(* Logix 5000 project; controller VET 1756-L62 rev 19.52; software revision 19.01; part 5 of 27 *)

        [443].S.BITS1.10   // 110-ENF-001/2 LH
        [444].S.BITS1.0   // 110-ENF-001/2-1 Enable
        [444].S.BITS1.1   // 110-ENF-001/2-1 Falla Resumen
        [444].S.BITS1.2   // 110-ENF-001/2-1 Conf. Marcha
        [444].S.BITS1.4   // 110-ENF-001/2-1 Cmd. Automatico
        [444].S.BITS1.26   // 110-ENF-001/2-1 FLL
        [444].S.BITS1.28   // 110-ENF-001/2-1 FATO
        [444].S.BITS1.30   // 110-ENF-001/2-1 Falla Partida
        [444].S.BITS2.27   // 110-ENF-001/2-1 Cmd. Marcha
        [444].S.BITS2.20   // 110-ENF-001/2-1 Reset Falla
        [444].S.BITS2.23   // 110-ENF-001/2-1 Test
        [444].S.BITS2.30   // 110-ENF-001/2-1 OUT MARCHA
        [447].S.BITS1.27   // 110-ESC-003/2 FV0
        [446].S.BITS1.8   // 9-BIN-708 LL
        [446].S.BITS1.9   // 9-BIN-708 LM
        [446].S.BITS1.10   // 9-BIN-708 LH
        [447].S.BITS1.0   // 9-CON-709 Enable
        [447].S.BITS1.1   // 9-CON-709 Falla Resumen
        [447].S.BITS1.26   // 110-ESC-003/2 FLL
        [447].S.BITS1.28   // 110-ESC-003/2 FATO
        [447].S.BITS2.20   // 9-CON-709 Reset Falla
        [447].S.BITS2.23   // 9-CON-709 Test
        [447].S.BITS2.30   // 9-CON-709 OUT CLOSE
        [449].S.BITS1.0   // 9-CON-711 Enable
        [449].S.BITS1.1   // 9-CON-711 Falla Resumen
        [449].S.BITS1.4   // 9-CON-711 Conf Pos Cerrar
        [449].S.BITS1.26   // 110-VAL-001/2-1 FLL
        [449].S.BITS1.27   // 110-VAL-001/2-1 FV0
        [449].S.BITS1.28   // 110-VAL-001/2-1 FATO
        [449].S.BITS2.20   // 9-CON-711 Reset Falla
        [449].S.BITS2.23   // 9-CON-711 Test
        [449].S.BITS2.30   // 9-CON-711 OUT CLOSE
        [450].S.BITS1.0   // 110-VEN-001/2 Enable
        [450].S.BITS1.1   // 110-VEN-001/2 Falla Resumen
        [450].S.BITS1.2   // 110-VEN-001/2 Conf. Marcha
        [450].S.BITS1.4   // 110-VEN-001/2 Cmd. Automatico
        [450].S.BITS1.26   // 110-VEN-001/2 FLL
        [450].S.BITS1.27   // 110-VEN-001/2 FV0
        [450].S.BITS1.28   // 110-VEN-001/2 FATO
        [450].S.BITS1.30   // 110-VEN-001/2 Falla Partida
        [450].S.BITS2.27   // 110-VEN-001/2 Cmd. Marcha
        [450].S.BITS2.20   // 110-VEN-001/2 Reset Falla
        [450].S.BITS2.23   // 110-VEN-001/2 Test
        [450].S.BITS2.30   // 110-VEN-001/2 OUT MARCHA
        [451].S.BITS1.0   // 9-CON-713 Enable
        [451].S.BITS1.1   // 9-CON-713 Falla Resumen
        [451].S.BITS1.2   // 9-CON-713 Conf Pos Abrir
        [451].S.BITS1.4   // 9-CON-713 Conf Pos Cerrar
        [451].S.BITS1.26   // 110-ENF-001/2-5 FLL
        [451].S.BITS1.27   // 110-ENF-001/2-5 FV0
        [451].S.BITS1.28   // 110-ENF-001/2-5 FATO
        [451].S.BITS1.30   // 9-CON-713 Falla Cerrar
        [451].S.BITS2.27   // 9-CON-713 Cmd. Open
        [451].S.BITS2.20   // 9-CON-713 Reset Falla
        [451].S.BITS2.23   // 9-CON-713 Test
        [451].S.BITS2.30   // 9-CON-713 OUT CLOSE
        [461].S.BITS1.0   // 9-CON-723 Enable
        [461].S.BITS1.1   // 9-CON-723 Falla Resumen
        [461].S.BITS1.2   // 9-CON-723 Conf Pos Abrir
        [461].S.BITS1.4   // 9-CON-723 Conf Pos Cerrar
        [461].S.BITS1.26   // 110-ESC-002/2 FLL
        [461].S.BITS1.27   // 110-ESC-002/2 FV0
        [461].S.BITS1.28   // 110-ESC-002/2 FATO
        [461].S.BITS1.30   // 9-CON-723 Falla Cerrar
        [461].S.BITS2.27   // 9-CON-723 Cmd. Open
        [461].S.BITS2.20   // 9-CON-723 Reset Falla
        [461].S.BITS2.23   // 9-CON-723 Test
        [461].S.BITS2.30   // 9-CON-723 OUT CLOSE
        [462].S.BITS1.0   // 110-ENF-002/2-4 Enable
        [462].S.BITS1.1   // 110-ENF-002/2-4 Falla Resumen
        [462].S.BITS1.2   // 110-ENF-002/2-4 Conf. Marcha
        [462].S.BITS1.4   // 110-ENF-002/2-4 Cmd. Automatico
        [462].S.BITS1.26   // 110-ENF-002/2-4 FLL
        [462].S.BITS1.27   // 110-ENF-002/2-4 FV0
        [462].S.BITS1.28   // 110-ENF-002/2-4 FATO
        [462].S.BITS1.30   // 110-ENF-002/2-4 Falla Partida
        [462].S.BITS2.27   // 110-ENF-002/2-4 Cmd. Marcha
        [462].S.BITS2.20   // 110-ENF-002/2-4 Reset Falla
        [462].S.BITS2.23   // 110-ENF-002/2-4 Test
        [462].S.BITS2.30   // 110-ENF-002/2-4 OUT MARCHA
        [464].S.BITS1.27   // 110-ENF-002/2-1 FV0
        [463].S.BITS1.8   // 110-ENF-002/2 LL
        [463].S.BITS1.9   // 110-ENF-002/2 LM
        [463].S.BITS1.10   // 110-ENF-002/2 LH
        [464].S.BITS1.0   // 110-ENF-002/2-1 Enable
        [464].S.BITS1.1   // 110-ENF-002/2-1 Falla Resumen
        [464].S.BITS1.2   // 110-ENF-002/2-1 Conf. Marcha
        [464].S.BITS1.4   // 110-ENF-002/2-1 Cmd. Automatico
        [464].S.BITS1.26   // 110-ENF-002/2-1 FLL
        [464].S.BITS1.28   // 110-ENF-002/2-1 FATO
        [464].S.BITS1.30   // 110-ENF-002/2-1 Falla Partida
        [464].S.BITS2.27   // 110-ENF-002/2-1 Cmd. Marcha
        [464].S.BITS2.20   // 110-ENF-002/2-1 Reset Falla
        [464].S.BITS2.23   // 110-ENF-002/2-1 Test
        [464].S.BITS2.30   // 110-ENF-002/2-1 OUT MARCHA
        [467].S.BITS1.27   // 110-ESC-004/2 FV0
        [466].S.BITS1.8   // 9-BIN-728 LL
        [466].S.BITS1.9   // 9-BIN-728 LM
        [466].S.BITS1.10   // 9-BIN-728 LH
        [467].S.BITS1.0   // 9-CON-729 Enable
        [467].S.BITS1.1   // 9-CON-729 Falla Resumen
        [467].S.BITS1.2   // 9-CON-729 Conf Pos Abrir
        [467].S.BITS1.4   // 9-CON-729 Conf Pos Cerrar
        [467].S.BITS1.26   // 110-ESC-004/2 FLL
        [467].S.BITS1.28   // 110-ESC-004/2 FATO
        [467].S.BITS1.30   // 9-CON-729 Falla Cerrar
        [467].S.BITS2.27   // 9-CON-729 Cmd. Open
        [467].S.BITS2.20   // 9-CON-729 Reset Falla
        [467].S.BITS2.23   // 9-CON-729 Test
        [467].S.BITS2.30   // 9-CON-729 OUT CLOSE
        [469].S.BITS1.0   // 9-CON-731 Enable
        [469].S.BITS1.1   // 9-CON-731 Falla Resumen
        [469].S.BITS1.2   // 9-CON-731 Conf Pos Abrir
        [469].S.BITS1.4   // 9-CON-731 Conf Pos Cerrar
        [469].S.BITS1.26   // 110-VAL-002/2-1 FLL
        [469].S.BITS1.27   // 110-VAL-002/2-1 FV0
        [469].S.BITS1.28   // 110-VAL-002/2-1 FATO
        [469].S.BITS1.30   // 9-CON-731 Falla Cerrar
        [469].S.BITS2.27   // 9-CON-731 Cmd. Open
        [469].S.BITS2.20   // 9-CON-731 Reset Falla
        [469].S.BITS2.23   // 9-CON-731 Test
        [469].S.BITS2.30   // 9-CON-731 OUT CLOSE
        [470].S.BITS1.0   // 110-VEN-002/2 Enable
        [470].S.BITS1.1   // 110-VEN-002/2 Falla Resumen
        [470].S.BITS1.2   // 110-VEN-002/2 Conf. Marcha
        [470].S.BITS1.4   // 110-VEN-002/2 Cmd. Automatico
        [470].S.BITS1.26   // 110-VEN-002/2 FLL
        [470].S.BITS1.27   // 110-VEN-002/2 FV0
        [470].S.BITS1.28   // 110-VEN-002/2 FATO
        [470].S.BITS1.30   // 110-VEN-002/2 Falla Partida
        [470].S.BITS2.27   // 110-VEN-002/2 Cmd. Marcha
        [470].S.BITS2.20   // 110-VEN-002/2 Reset Falla
        [470].S.BITS2.23   // 110-VEN-002/2 Test
        [470].S.BITS2.30   // 110-VEN-002/2 OUT MARCHA
        [471].S.BITS1.0   // 110-ENF-002/2-5 Enable
        [471].S.BITS1.1   // 110-ENF-002/2-5 Falla Resumen
        [471].S.BITS1.2   // 110-ENF-002/2-5 Conf. Marcha
        [471].S.BITS1.4   // 110-ENF-002/2-5 Cmd. Automatico
        [471].S.BITS1.26   // 110-ENF-002/2-5 FLL
        [471].S.BITS1.27   // 110-ENF-002/2-5 FV0
        [471].S.BITS1.28   // 110-ENF-002/2-5 FATO
        [471].S.BITS1.30   // 110-ENF-002/2-5 Falla Partida
        [471].S.BITS2.27   // 110-ENF-002/2-5 Cmd. Marcha
        [471].S.BITS2.20   // 110-ENF-002/2-5 Reset Falla
        [471].S.BITS2.23   // 110-ENF-002/2-5 Test
        [471].S.BITS2.30   // 110-ENF-002/2-5 OUT MARCHA
        [474].S.BITS1.0   // 110-TOR-002/2 Enable
        [474].S.BITS1.1   // 110-TOR-002/2 Falla Resumen
        [474].S.BITS1.26   // 110-TOR-002/2 FLL
        [474].S.BITS1.27   // 110-TOR-002/2 FV0
        [474].S.BITS1.28   // 110-TOR-002/2 FATO
        [474].S.BITS2.20   // 110-TOR-002/2 Reset Falla
        [474].S.BITS2.23   // 110-TOR-002/2 Test
        [474].S.BITS2.30   // 110-TOR-002/2 OUT MARCHA
        [475].S.BITS1.0   // 110-TOR-003/2 Enable
        [475].S.BITS1.1   // 110-TOR-003/2 Falla Resumen
        [475].S.BITS1.26   // 110-TOR-003/2 FLL
        [475].S.BITS1.27   // 110-TOR-003/2 FV0
        [475].S.BITS1.28   // 110-TOR-003/2 FATO
        [475].S.BITS2.20   // 110-TOR-003/2 Reset Falla
        [475].S.BITS2.23   // 110-TOR-003/2 Test
        [475].S.BITS2.30   // 110-TOR-003/2 OUT MARCHA
        [476].S.BITS1.0   // 110-ELV-002/2 Enable
        [476].S.BITS1.1   // 110-ELV-002/2 Falla Resumen
        [476].S.BITS1.26   // 110-ELV-002/2 FLL
        [476].S.BITS1.27   // 110-ELV-002/2 FV0
        [476].S.BITS1.28   // 110-ELV-002/2 FATO
        [476].S.BITS2.20   // 110-ELV-002/2 Reset Falla
        [476].S.BITS2.23   // 110-ELV-002/2 Test
        [478].S.BITS1.27   // 110-TOR-004/2 FV0
        [477].S.BITS1.8   // 110-TOL-006/2 LL
        [477].S.BITS1.9   // 110-TOL-006/2 LM
        [477].S.BITS1.10   // 110-TOL-006/2 LH
        [478].S.BITS1.0   // 110-TOR-004/2 Enable
        [478].S.BITS1.1   // 110-TOR-004/2 Falla Resumen
        [478].S.BITS1.2   // 110-TOR-004/2 Conf. Marcha
        [478].S.BITS1.4   // 110-TOR-004/2 Cmd. Automatico
        [478].S.BITS1.26   // 110-TOR-004/2 FLL
        [478].S.BITS1.28   // 110-TOR-004/2 FATO
        [478].S.BITS1.30   // 110-TOR-004/2 Falla Partida
        [478].S.BITS2.27   // 110-TOR-004/2 Cmd. Marcha
        [478].S.BITS2.20   // 110-TOR-004/2 Reset Falla
        [478].S.BITS2.23   // 110-TOR-004/2 Test
        [478].S.BITS2.30   // 110-TOR-004/2 OUT MARCHA
        [493].S.BITS1.1   // 110-CAN-008/3 Falla Resumen
        [491].S.BITS1.8   // 110-TOL-005/3 LL
        [491].S.BITS1.9   // 110-TOL-005/3 LM
        [491].S.BITS1.10   // 110-TOL-005/3 LH
        [493].S.BITS1.30   // 110-CAN-008/3 Falla Cerrar
        [492].S.BITS1.8   // 110-TOL-004/3 LL
        [492].S.BITS1.9   // 110-TOL-004/3 LM
        [492].S.BITS1.10   // 110-TOL-004/3 LH
        [493].S.BITS1.0   // 110-CAN-008/3 Enable
        [493].S.BITS1.2   // 110-CAN-008/3 Conf Pos Abrir
        [493].S.BITS1.4   // 110-CAN-008/3 Conf Pos Cerrar
        [493].S.BITS1.29   // 110-CAN-008/3 Falla Abrir
        [493].S.BITS2.20   // 110-CAN-008/3 Reset Falla
        [493].S.BITS2.23   // 110-CAN-008/3 Test
        [493].S.BITS2.27   // 110-CAN-008/3 Cmd. Open
        [493].S.BITS2.30   // 110-CAN-008/3 OUT CLOSE
        [493].S.BITS2.31   // 110-CAN-008/3 OUT OPEN
        [494].S.BITS1.0   // 110-CAN-009/3 Enable
        [494].S.BITS1.1   // 110-CAN-009/3 Falla Resumen
        [494].S.BITS1.2   // 110-CAN-009/3 Conf Pos Abrir
        [494].S.BITS1.4   // 110-CAN-009/3 Conf Pos Cerrar
        [494].S.BITS1.29   // 110-CAN-009/3 Falla Abrir
        [494].S.BITS1.30   // 110-CAN-009/3 Falla Cerrar
        [494].S.BITS2.20   // 110-CAN-009/3 Reset Falla
        [494].S.BITS2.23   // 110-CAN-009/3 Test
        [494].S.BITS2.27   // 110-CAN-009/3 Cmd. Open
        [494].S.BITS2.30   // 110-CAN-009/3 OUT CLOSE
        [494].S.BITS2.31   // 110-CAN-009/3 OUT OPEN
        [495].S.BITS1.0   // 110-CAN-010/3 Enable
        [495].S.BITS1.1   // 110-CAN-010/3 Falla Resumen
        [495].S.BITS1.2   // 110-CAN-010/3 Conf. Marcha
        [495].S.BITS1.4   // 110-CAN-010/3 Cmd. Automatico
        [495].S.BITS1.26   // 110-CAN-010/3 FLL
        [495].S.BITS1.27   // 110-CAN-010/3 FV0
        [495].S.BITS1.28   // 110-CAN-010/3 FATO
        [495].S.BITS1.30   // 110-CAN-010/3 Falla Partida
        [495].S.BITS2.27   // 110-CAN-010/3 Cmd. Marcha
        [495].S.BITS2.20   // 110-CAN-010/3 Reset Falla
        [495].S.BITS2.23   // 110-CAN-010/3 Test
        [495].S.BITS2.30   // 110-CAN-010/3 OUT MARCHA
        [497].S.BITS1.30   // 110-CAN-011/3 Falla Cerrar
        [496].S.BITS1.8   // 110-TOL-006/3 LL
        [496].S.BITS1.9   // 110-TOL-006/3 LM
        [496].S.BITS1.10   // 110-TOL-006/3 LH
        [497].S.BITS1.0   // 110-CAN-011/3 Enable
        [497].S.BITS1.1   // 110-CAN-011/3 Falla Resumen
        [497].S.BITS1.2   // 110-CAN-011/3 Conf Pos Abrir
        [497].S.BITS1.4   // 110-CAN-011/3 Conf Pos Cerrar
        [497].S.BITS1.29   // 110-CAN-011/3 Falla Abrir
        [497].S.BITS2.20   // 110-CAN-011/3 Reset Falla
        [497].S.BITS2.23   // 110-CAN-011/3 Test
        [497].S.BITS2.27   // 110-CAN-011/3 Cmd. Open
        [497].S.BITS2.30   // 110-CAN-011/3 OUT CLOSE
        [497].S.BITS2.31   // 110-CAN-011/3 OUT OPEN
        [500].S.BITS1.27   // 110-TOR-001/3 FV0
        [499].S.BITS1.8   // 110-TOL-007/3 LL
        [499].S.BITS1.9   // 110-TOL-007/3 LM
        [499].S.BITS1.10   // 110-TOL-007/3 LH
        [500].S.BITS1.0   // 110-TOR-001/3 Enable
        [500].S.BITS1.1   // 110-TOR-001/3 Falla Resumen
        [500].S.BITS1.2   // 110-TOR-001/3 Conf. Marcha
        [500].S.BITS1.4   // 110-TOR-001/3 Cmd. Automatico
        [500].S.BITS1.26   // 110-TOR-001/3 FLL
        [500].S.BITS1.28   // 110-TOR-001/3 FATO
        [500].S.BITS1.30   // 110-TOR-001/3 Falla Partida
        [500].S.BITS2.27   // 110-TOR-001/3 Cmd. Marcha
        [500].S.BITS2.20   // 110-TOR-001/3 Reset Falla
        [500].S.BITS2.23   // 110-TOR-001/3 Test
        [500].S.BITS2.30   // 110-TOR-001/3 OUT MARCHA
        [502].S.BITS1.0   // 110-ACD-001/3 Enable
        [502].S.BITS1.1   // 110-ACD-001/3 Falla Resumen
        [502].S.BITS1.2   // 110-ACD-001/3 Conf. Marcha
        [502].S.BITS1.4   // 110-ACD-001/3 Cmd. Automatico
        [502].S.BITS1.26   // 110-ACD-001/3 FLL
        [502].S.BITS1.27   // 110-ACD-001/3 FV0
        [502].S.BITS1.28   // 110-ACD-001/3 FATO
        [502].S.BITS1.30   // 110-ACD-001/3 Falla Partida
        [502].S.BITS2.27   // 110-ACD-001/3 Cmd. Marcha
        [502].S.BITS2.20   // 110-ACD-001/3 Reset Falla
        [502].S.BITS2.23   // 110-ACD-001/3 Test
        [502].S.BITS2.30   // 110-ACD-001/3 OUT MARCHA
        [503].S.BITS1.0   // 110-EXP-001/3 Enable
        [503].S.BITS1.1   // 110-EXP-001/3 Falla Resumen
        [503].S.BITS1.4   // 110-EXP-001/3 Cmd. Automatico
        [503].S.BITS1.26   // 110-EXP-001/3 FLL
        [503].S.BITS1.27   // 110-EXP-001/3 FV0
        [503].S.BITS1.28   // 110-EXP-001/3 FATO
        [503].S.BITS1.30   // 110-EXP-001/3 Falla Partida
        [503].S.BITS2.27   // 110-EXP-001/3 Cmd. Marcha
        [503].S.BITS2.20   // 110-EXP-001/3 Reset Falla
        [503].S.BITS2.23   // 110-EXP-001/3 Test
        [503].S.BITS2.30   // 110-EXP-001/3 OUT MARCHA
        [504].S.BITS1.0   // 110-DES-001/3 Enable
        [504].S.BITS1.1   // 110-DES-001/3 Falla Resumen
        [504].S.BITS1.2   // 110-DES-001/3 Conf. Marcha
        [504].S.BITS1.4   // 110-DES-001/3 Cmd. Automatico
        [504].S.BITS1.26   // 110-DES-001/3 FLL
        [504].S.BITS1.27   // 110-DES-001/3 FV0
        [504].S.BITS1.28   // 110-DES-001/3 FATO
        [504].S.BITS1.30   // 110-DES-001/3 Falla Partida
        [504].S.BITS2.27   // 110-DES-001/3 Cmd. Marcha
        [504].S.BITS2.20   // 110-DES-001/3 Reset Falla
        [504].S.BITS2.23   // 110-DES-001/3 Test
        [504].S.BITS2.30   // 110-DES-001/3 OUT MARCHA
        [505].S.BITS1.0   // 110-CAE-001/3 Enable
        [505].S.BITS1.1   // 110-CAE-001/3 Falla Resumen
        [505].S.BITS1.2   // 110-CAE-001/3 Conf. Marcha
        [505].S.BITS1.4   // 110-CAE-001/3 Cmd. Automatico
        [505].S.BITS1.26   // 110-CAE-001/3 FLL
        [505].S.BITS1.27   // 110-CAE-001/3 FV0
        [505].S.BITS1.28   // 110-CAE-001/3 FATO
        [505].S.BITS1.30   // 110-CAE-001/3 Falla Partida
        [505].S.BITS2.27   // 110-CAE-001/3 Cmd. Marcha
        [505].S.BITS2.20   // 110-CAE-001/3 Reset Falla
        [505].S.BITS2.23   // 110-CAE-001/3 Test
        [505].S.BITS2.30   // 110-CAE-001/3 OUT MARCHA
        [506].S.BITS1.0   // 110-PLT-001/3 Enable
        [506].S.BITS1.1   // 110-PLT-001/3 Falla Resumen
        [506].S.BITS1.2   // 110-PLT-001/3 Conf. Marcha
        [506].S.BITS1.4   // 110-PLT-001/3 Cmd. Automatico
        [506].S.BITS1.26   // 110-PLT-001/3 FLL
        [506].S.BITS1.27   // 110-PLT-001/3 FV0
        [506].S.BITS1.28   // 110-PLT-001/3 FATO
        [506].S.BITS1.30   // 110-PLT-001/3 Falla Partida
        [506].S.BITS2.27   // 110-PLT-001/3 Cmd. Marcha
        [506].S.BITS2.20   // 110-PLT-001/3 Reset Falla
        [506].S.BITS2.23   // 110-PLT-001/3 Test
        [506].S.BITS2.30   // 110-PLT-001/3 OUT MARCHA
        [507].S.BITS1.0   // 110-BIF-001/3 Enable
        [507].S.BITS1.1   // 110-BIF-001/3 Falla Resumen
        [507].S.BITS1.2   // 110-BIF-001/3 Conf. Pos. Izquierda
        [507].S.BITS1.4   // 110-BIF-001/3 Conf. Pos. Derecha
        [507].S.BITS1.29   // 110-BIF-001/3 Falla Pos. Izquierda
        [507].S.BITS1.30   // 110-BIF-001/3 Falla Pos. Derecha
        [507].S.BITS2.20   // 110-BIF-001/3 Reset Falla
        [507].S.BITS2.23   // 110-BIF-001/3 Test
        [507].S.BITS2.26   // 110-BIF-001/3 Cmd. Pos . Izquierda
        [507].S.BITS2.27   // 110-BIF-001/3 Cmd. Pos. Derecha
        [507].S.BITS2.30   // 110-BIF-001/3 Out Izquierda
        [507].S.BITS2.31   // 110-BIF-001/3 Out Derecha
        [511].S.BITS1.0   // 110-ESC-001/3 Enable
        [511].S.BITS1.1   // 110-ESC-001/3 Falla Resumen
        [511].S.BITS1.2   // 110-ESC-001/3 Conf. Marcha
        [511].S.BITS1.4   // 110-ESC-001/3 Cmd. Automatico
        [511].S.BITS1.26   // 110-ESC-001/3 FLL
        [511].S.BITS1.27   // 110-ESC-001/3 FV0
        [511].S.BITS1.28   // 110-ESC-001/3 FATO
        [511].S.BITS1.30   // 110-ESC-001/3 Falla Partida
        [511].S.BITS2.27   // 110-ESC-001/3 Cmd. Marcha
        [511].S.BITS2.20   // 110-ESC-001/3 Reset Falla
        [511].S.BITS2.23   // 110-ESC-001/3 Test
        [511].S.BITS2.30   // 110-ESC-001/3 OUT MARCHA
        [512].S.BITS1.0   // 110-ENF-001/3-4 Enable
        [512].S.BITS1.1   // 110-ENF-001/3-4 Falla Resumen
        [512].S.BITS1.2   // 110-ENF-001/3-4 Conf. Marcha
        [512].S.BITS1.4   // 110-ENF-001/3-4 Cmd. Automatico
        [512].S.BITS1.26   // 110-ENF-001/3-4 FLL
        [512].S.BITS1.27   // 110-ENF-001/3-4 FV0
        [512].S.BITS1.28   // 110-ENF-001/3-4 FATO
        [512].S.BITS1.30   // 110-ENF-001/3-4 Falla Partida
        [512].S.BITS2.27   // 110-ENF-001/3-4 Cmd. Marcha
        [512].S.BITS2.20   // 110-ENF-001/3-4 Reset Falla
        [512].S.BITS2.23   // 110-ENF-001/3-4 Test
        [512].S.BITS2.30   // 110-ENF-001/3-4 OUT MARCHA
        [514].S.BITS1.27   // 110-ENF-001/3-1 FV0
        [513].S.BITS1.8   // 110-ENF-001/3 LL
        [513].S.BITS1.9   // 110-ENF-001/3 LM
        [513].S.BITS1.10   // 110-ENF-001/3 LH
        [514].S.BITS1.0   // 110-ENF-001/3-1 Enable
        [514].S.BITS1.1   // 110-ENF-001/3-1 Falla Resumen
        [514].S.BITS1.2   // 110-ENF-001/3-1 Conf. Marcha
        [514].S.BITS1.4   // 110-ENF-001/3-1 Cmd. Automatico
        [514].S.BITS1.26   // 110-ENF-001/3-1 FLL
        [514].S.BITS1.28   // 110-ENF-001/3-1 FATO
        [514].S.BITS1.30   // 110-ENF-001/3-1 Falla Partida
        [514].S.BITS2.27   // 110-ENF-001/3-1 Cmd. Marcha
        [514].S.BITS2.20   // 110-ENF-001/3-1 Reset Falla
        [514].S.BITS2.23   // 110-ENF-001/3-1 Test
        [514].S.BITS2.30   // 110-ENF-001/3-1 OUT MARCHA
        [517].S.BITS1.27   // 110-ESC-003/3 FV0
        [516].S.BITS1.8   // 110-CIC-001/3 LL
        [516].S.BITS1.9   // 110-CIC-001/3 LM
        [516].S.BITS1.10   // 110-CIC-001/3 LH
        [517].S.BITS1.0   // 110-ESC-003/3 Enable
        [517].S.BITS1.1   // 110-ESC-003/3 Falla Resumen
        [517].S.BITS1.2   // 110-ESC-003/3 Conf. Marcha
        [517].S.BITS1.4   // 110-ESC-003/3 Cmd. Automatico
        [517].S.BITS1.26   // 110-ESC-003/3 FLL
        [517].S.BITS1.28   // 110-ESC-003/3 FATO
        [517].S.BITS1.30   // 110-ESC-003/3 Falla Partida
        [517].S.BITS2.27   // 110-ESC-003/3 Cmd. Marcha
        [517].S.BITS2.20   // 110-ESC-003/3 Reset Falla
        [517].S.BITS2.23   // 110-ESC-003/3 Test
        [517].S.BITS2.30   // 110-ESC-003/3 OUT MARCHA
        [519].S.BITS1.0   // 110-VAL-001/3-1 Enable
        [519].S.BITS1.1   // 110-VAL-001/3-1 Falla Resumen
        [519].S.BITS1.2   // 110-VAL-001/3-1 Conf. Marcha
        [519].S.BITS1.4   // 110-VAL-001/3-1 Cmd. Automatico
        [519].S.BITS1.26   // 110-VAL-001/3-1 FLL
        [519].S.BITS1.27   // 110-VAL-001/3-1 FV0
        [519].S.BITS1.28   // 110-VAL-001/3-1 FATO
        [519].S.BITS1.30   // 110-VAL-001/3-1 Falla Partida
        [519].S.BITS2.27   // 110-VAL-001/3-1 Cmd. Marcha
        [519].S.BITS2.20   // 110-VAL-001/3-1 Reset Falla
        [519].S.BITS2.23   // 110-VAL-001/3-1 Test
        [519].S.BITS2.30   // 110-VAL-001/3-1 OUT MARCHA
        [520].S.BITS1.0   // 110-VEN-001/3 Enable
        [520].S.BITS1.1   // 110-VEN-001/3 Falla Resumen
        [520].S.BITS1.2   // 110-VEN-001/3 Conf. Marcha
        [520].S.BITS1.4   // 110-VEN-001/3 Cmd. Automatico
        [520].S.BITS1.26   // 110-VEN-001/3 FLL
        [520].S.BITS1.27   // 110-VEN-001/3 FV0
        [520].S.BITS1.28   // 110-VEN-001/3 FATO
        [520].S.BITS1.30   // 110-VEN-001/3 Falla Partida
        [520].S.BITS2.27   // 110-VEN-001/3 Cmd. Marcha
        [520].S.BITS2.20   // 110-VEN-001/3 Reset Falla
        [520].S.BITS2.23   // 110-VEN-001/3 Test
        [520].S.BITS2.30   // 110-VEN-001/3 OUT MARCHA
        [521].S.BITS1.0   // 110-ENF-001/3-5 Enable
        [521].S.BITS1.1   // 110-ENF-001/3-5 Falla Resumen
        [521].S.BITS1.2   // 110-ENF-001/3-5 Conf. Marcha
        [521].S.BITS1.4   // 110-ENF-001/3-5 Cmd. Automatico
        [521].S.BITS1.26   // 110-ENF-001/3-5 FLL
        [521].S.BITS1.27   // 110-ENF-001/3-5 FV0
        [521].S.BITS1.28   // 110-ENF-001/3-5 FATO
        [521].S.BITS1.30   // 110-ENF-001/3-5 Falla Partida
        [521].S.BITS2.27   // 110-ENF-001/3-5 Cmd. Marcha
        [521].S.BITS2.20   // 110-ENF-001/3-5 Reset Falla
        [521].S.BITS2.23   // 110-ENF-001/3-5 Test
        [521].S.BITS2.30   // 110-ENF-001/3-5 OUT MARCHA
        [523].S.BITS1.0   // 110-QUE-001-1 Enable
        [523].S.BITS1.1   // 110-QUE-001-1 Falla Resumen
        [523].S.BITS1.2   // 110-QUE-001-1 Conf. Marcha
        [523].S.BITS1.4   // 110-QUE-001-1 Cmd. Automatico
        [523].S.BITS1.26   // 110-QUE-001-1 FLL
        [523].S.BITS1.27   // 110-QUE-001-1 FV0
        [523].S.BITS1.28   // 110-QUE-001-1 FATO
        [523].S.BITS1.30   // 110-QUE-001-1 Falla Partida
        [523].S.BITS2.27   // 110-QUE-001-1 Cmd. Marcha
        [523].S.BITS2.20   // 110-QUE-001-1 Reset Falla
        [523].S.BITS2.23   // 110-QUE-001-1 Test
        [523].S.BITS2.30   // 110-QUE-001-1 OUT MARCHA
        [524].S.BITS1.0   // 110-QUE-001-2 Enable
        [524].S.BITS1.1   // 110-QUE-001-2 Falla Resumen
        [524].S.BITS1.2   // 110-QUE-001-2 Conf. Marcha
        [524].S.BITS1.4   // 110-QUE-001-2 Cmd. Automatico
        [524].S.BITS1.26   // 110-QUE-001-2 FLL
        [524].S.BITS1.27   // 110-QUE-001-2 FV0
        [524].S.BITS1.28   // 110-QUE-001-2 FATO
        [524].S.BITS1.30   // 110-QUE-001-2 Falla Partida
        [524].S.BITS2.27   // 110-QUE-001-2 Cmd. Marcha
        [524].S.BITS2.20   // 110-QUE-001-2 Reset Falla
        [524].S.BITS2.23   // 110-QUE-001-2 Test
        [524].S.BITS2.30   // 110-QUE-001-2 OUT MARCHA
        [531].S.BITS1.0   // 110-ESC-002/3 Enable
        [531].S.BITS1.1   // 110-ESC-002/3 Falla Resumen
        [531].S.BITS1.2   // 110-ESC-002/3 Conf. Marcha
        [531].S.BITS1.4   // 110-ESC-002/3 Cmd. Automatico
        [531].S.BITS1.26   // 110-ESC-002/3 FLL
        [531].S.BITS1.27   // 110-ESC-002/3 FV0
        [531].S.BITS1.28   // 110-ESC-002/3 FATO
        [531].S.BITS1.30   // 110-ESC-002/3 Falla Partida
        [531].S.BITS2.27   // 110-ESC-002/3 Cmd. Marcha
        [531].S.BITS2.20   // 110-ESC-002/3 Reset Falla
        [531].S.BITS2.23   // 110-ESC-002/3 Test
        [531].S.BITS2.30   // 110-ESC-002/3 OUT MARCHA
        [532].S.BITS1.0   // 110-ENF-002/3-4 Enable
        [532].S.BITS1.1   // 110-ENF-002/3-4 Falla Resumen
        [532].S.BITS1.2   // 110-ENF-002/3-4 Conf. Marcha
        [532].S.BITS1.4   // 110-ENF-002/3-4 Cmd. Automatico
        [532].S.BITS1.26   // 110-ENF-002/3-4 FLL
        [532].S.BITS1.27   // 110-ENF-002/3-4 FV0
        [532].S.BITS1.28   // 110-ENF-002/3-4 FATO
        [532].S.BITS1.30   // 110-ENF-002/3-4 Falla Partida
        [532].S.BITS2.27   // 110-ENF-002/3-4 Cmd. Marcha
        [532].S.BITS2.20   // 110-ENF-002/3-4 Reset Falla
        [532].S.BITS2.23   // 110-ENF-002/3-4 Test
        [532].S.BITS2.30   // 110-ENF-002/3-4 OUT MARCHA
        [534].S.BITS1.27   // 110-ENF-002/3-1 FV0
        [533].S.BITS1.8   // 110-ENF-002/3 LL
        [533].S.BITS1.9   // 110-ENF-002/3 LM
        [533].S.BITS1.10   // 110-ENF-002/3 LH
        [534].S.BITS1.0   // 110-ENF-002/3-1 Enable
        [534].S.BITS1.1   // 110-ENF-002/3-1 Falla Resumen
        [534].S.BITS1.2   // 110-ENF-002/3-1 Conf. Marcha
        [534].S.BITS1.4   // 110-ENF-002/3-1 Cmd. Automatico
        [534].S.BITS1.26   // 110-ENF-002/3-1 FLL
        [534].S.BITS1.28   // 110-ENF-002/3-1 FATO
        [534].S.BITS1.30   // 110-ENF-002/3-1 Falla Partida
        [534].S.BITS2.27   // 110-ENF-002/3-1 Cmd. Marcha
        [534].S.BITS2.20   // 110-ENF-002/3-1 Reset Falla
        [534].S.BITS2.23   // 110-ENF-002/3-1 Test
        [534].S.BITS2.30   // 110-ENF-002/3-1 OUT MARCHA
        [537].S.BITS1.27   // 110-ESC-004/3 FV0
        [536].S.BITS1.8   // 110-CIC-002/3 LL
        [536].S.BITS1.9   // 110-CIC-002/3 LM
        [536].S.BITS1.10   // 110-CIC-002/3 LH
        [537].S.BITS1.0   // 110-ESC-004/3 Enable
        [537].S.BITS1.1   // 110-ESC-004/3 Falla Resumen
        [537].S.BITS1.2   // 110-ESC-004/3 Conf. Marcha
        [537].S.BITS1.4   // 110-ESC-004/3 Cmd. Automatico
        [537].S.BITS1.26   // 110-ESC-004/3 FLL
        [537].S.BITS1.28   // 110-ESC-004/3 FATO
        [537].S.BITS1.30   // 110-ESC-004/3 Falla Partida
        [537].S.BITS2.27   // 110-ESC-004/3 Cmd. Marcha
        [537].S.BITS2.20   // 110-ESC-004/3 Reset Falla
        [537].S.BITS2.23   // 110-ESC-004/3 Test
        [537].S.BITS2.30   // 110-ESC-004/3 OUT MARCHA
        [539].S.BITS1.0   // 110-VEN-002/3-1 Enable
        [539].S.BITS1.1   // 110-VEN-002/3-1 Falla Resumen
        [539].S.BITS1.2   // 110-VEN-002/3-1 Conf. Marcha
        [539].S.BITS1.4   // 110-VEN-002/3-1 Cmd. Automatico
        [539].S.BITS1.26   // 110-VEN-002/3-1 FLL
        [539].S.BITS1.27   // 110-VEN-002/3-1 FV0
        [539].S.BITS1.28   // 110-VEN-002/3-1 FATO
        [539].S.BITS1.30   // 110-VEN-002/3-1 Falla Partida
        [539].S.BITS2.27   // 110-VEN-002/3-1 Cmd. Marcha
        [539].S.BITS2.20   // 110-VEN-002/3-1 Reset Falla
        [539].S.BITS2.23   // 110-VEN-002/3-1 Test
        [539].S.BITS2.30   // 110-VEN-002/3-1 OUT MARCHA
        [540].S.BITS1.0   // 110-VEN-002/3 Enable
        [540].S.BITS1.1   // 110-VEN-002/3 Falla Resumen
        [540].S.BITS1.2   // 110-VEN-002/3 Conf. Marcha
        [540].S.BITS1.4   // 110-VEN-002/3 Cmd. Automatico
        [540].S.BITS1.26   // 110-VEN-002/3 FLL
        [540].S.BITS1.27   // 110-VEN-002/3 FV0
        [540].S.BITS1.28   // 110-VEN-002/3 FATO
        [540].S.BITS1.30   // 110-VEN-002/3 Falla Partida
        [540].S.BITS2.27   // 110-VEN-002/3 Cmd. Marcha
        [540].S.BITS2.20   // 110-VEN-002/3 Reset Falla
        [540].S.BITS2.23   // 110-VEN-002/3 Test
        [540].S.BITS2.30   // 110-VEN-002/3 OUT MARCHA
        [541].S.BITS1.0   // 110-ENF-002/3-5 Enable
        [541].S.BITS1.1   // 110-ENF-002/3-5 Falla Resumen
        [541].S.BITS1.2   // 110-ENF-002/3-5 Conf. Marcha
        [541].S.BITS1.4   // 110-ENF-002/3-5 Cmd. Automatico
        [541].S.BITS1.26   // 110-ENF-002/3-5 FLL
        [541].S.BITS1.27   // 110-ENF-002/3-5 FV0
        [541].S.BITS1.28   // 110-ENF-002/3-5 FATO
        [541].S.BITS1.30   // 110-ENF-002/3-5 Falla Partida
        [541].S.BITS2.27   // 110-ENF-002/3-5 Cmd. Marcha
        [541].S.BITS2.20   // 110-ENF-002/3-5 Reset Falla
        [541].S.BITS2.23   // 110-ENF-002/3-5 Test
        [541].S.BITS2.30   // 110-ENF-002/3-5 OUT MARCHA
        [544].S.BITS1.0   // 110-TOR-002/3 Enable
        [544].S.BITS1.1   // 110-TOR-002/3 Falla Resumen
        [544].S.BITS1.2   // 110-TOR-002/3 Conf. Marcha
        [544].S.BITS1.4   // 110-TOR-002/3 Cmd. Automatico
        [544].S.BITS1.26   // 110-TOR-002/3 FLL
        [544].S.BITS1.27   // 110-TOR-002/3 FV0
        [544].S.BITS1.28   // 110-TOR-002/3 FATO
        [544].S.BITS1.30   // 110-TOR-002/3 Falla Partida
        [544].S.BITS2.27   // 110-TOR-002/3 Cmd. Marcha
        [544].S.BITS2.20   // 110-TOR-002/3 Reset Falla
        [544].S.BITS2.23   // 110-TOR-002/3 Test
        [544].S.BITS2.30   // 110-TOR-002/3 OUT MARCHA
        [545].S.BITS1.0   // 110-TOR-003/3 Enable
        [545].S.BITS1.1   // 110-TOR-003/3 Falla Resumen
        [545].S.BITS1.2   // 110-TOR-003/3 Conf. Marcha
        [545].S.BITS1.4   // 110-TOR-003/3 Cmd. Automatico
        [545].S.BITS1.26   // 110-TOR-003/3 FLL
        [545].S.BITS1.27   // 110-TOR-003/3 FV0
        [545].S.BITS1.28   // 110-TOR-003/3 FATO
        [545].S.BITS1.30   // 110-TOR-003/3 Falla Partida
        [545].S.BITS2.27   // 110-TOR-003/3 Cmd. Marcha
        [545].S.BITS2.20   // 110-TOR-003/3 Reset Falla
        [545].S.BITS2.23   // 110-TOR-003/3 Test
        [545].S.BITS2.30   // 110-TOR-003/3 OUT MARCHA
        [546].S.BITS1.0   // 110-ELV-002/3 Enable
        [546].S.BITS1.1   // 110-ELV-002/3 Falla Resumen
        [546].S.BITS1.2   // 110-ELV-002/3 Conf. Marcha
        [546].S.BITS1.4   // 110-ELV-002/3 Cmd. Automatico
        [546].S.BITS1.26   // 110-ELV-002/3 FLL
        [546].S.BITS1.27   // 110-ELV-002/3 FV0
        [546].S.BITS1.28   // 110-ELV-002/3 FATO
        [546].S.BITS1.30   // 110-ELV-002/3 Falla Partida
        [546].S.BITS2.27   // 110-ELV-002/3 Cmd. Marcha
        [546].S.BITS2.20   // 110-ELV-002/3 Reset Falla
        [546].S.BITS2.23   // 110-ELV-002/3 Test
        [546].S.BITS2.30   // 110-ELV-002/3 OUT MARCHA
        [548].S.BITS1.27   // 110-TOR-004/3 FV0
        [547].S.BITS1.8   // 110-TOL-008/3 LL
        [547].S.BITS1.9   // 110-TOL-008/3 LM
        [547].S.BITS1.10   // 110-TOL-008/3 LH
        [548].S.BITS1.0   // 110-TOR-004/3 Enable
        [548].S.BITS1.1   // 110-TOR-004/3 Falla Resumen
        [548].S.BITS1.2   // 110-TOR-004/3 Conf. Marcha
        [548].S.BITS1.4   // 110-TOR-004/3 Cmd. Automatico
        [548].S.BITS1.26   // 110-TOR-004/3 FLL
        [548].S.BITS1.28   // 110-TOR-004/3 FATO
        [548].S.BITS1.30   // 110-TOR-004/3 Falla Partida
        [548].S.BITS2.27   // 110-TOR-004/3 Cmd. Marcha
        [548].S.BITS2.20   // 110-TOR-004/3 Reset Falla
        [548].S.BITS2.23   // 110-TOR-004/3 Test
        [548].S.BITS2.30   // 110-TOR-004/3 OUT MARCHA
        [551].S.BITS1.0   // 110-TDC-003/1 Enable
        [551].S.BITS1.1   // 110-TDC-003/1 Falla Resumen
        [551].S.BITS1.2   // 110-TDC-003/1 Conf. Marcha
        [551].S.BITS1.4   // 110-TDC-003/1 Cmd. Automatico
        [551].S.BITS1.26   // 110-TDC-003/1 FLL
        [551].S.BITS1.27   // 110-TDC-003/1 FV0
        [551].S.BITS1.28   // 110-TDC-003/1 FATO
        [551].S.BITS1.30   // 110-TDC-003/1 Falla Partida
        [551].S.BITS2.27   // 110-TDC-003/1 Cmd. Marcha
        [551].S.BITS2.20   // 110-TDC-003/1 Reset Falla
        [551].S.BITS2.23   // 110-TDC-003/1 Test
        [551].S.BITS2.30   // 110-TDC-003/1 OUT MARCHA
        [552].S.BITS1.26   // 110-TDC-004/1 FLL
        [552].S.BITS1.27   // 110-TDC-004/1 FV0
        [552].S.BITS1.28   // 110-TDC-004/1 FATO
        [554].S.BITS1.26   // 110-ELV-001/1 FLL
        [554].S.BITS1.27   // 110-ELV-001/1 FV0
        [554].S.BITS1.28   // 110-ELV-001/1 FATO
        [555].S.BITS1.0   // 120-TDC-001/1 Enable
        [555].S.BITS1.1   // 120-TDC-001/1 Falla Resumen
        [555].S.BITS1.2   // 120-TDC-001/1 Conf. Marcha
        [555].S.BITS1.4   // 120-TDC-001/1 Cmd. Automatico
        [555].S.BITS1.26   // 120-TDC-001/1 FLL
        [555].S.BITS1.27   // 120-TDC-001/1 FV0
        [555].S.BITS1.28   // 120-TDC-001/1 FATO
        [555].S.BITS1.30   // 120-TDC-001/1 Falla Partida
        [555].S.BITS2.27   // 120-TDC-001/1 Cmd. Marcha
        [555].S.BITS2.20   // 120-TDC-001/1 Reset Falla
        [555].S.BITS2.23   // 120-TDC-001/1 Test
        [555].S.BITS2.30   // 120-TDC-001/1 OUT MARCHA
        [556].S.BITS1.26   // 120-HAR-001 FLL
        [556].S.BITS1.27   // 120-HAR-001 FV0
        [556].S.BITS1.28   // 120-HAR-001 FATO
        [557].S.BITS1.0   // 120-XY-8127 Enable
        [557].S.BITS1.1   // 120-XY-8127 Falla Resumen
        [557].S.BITS1.2   // 120-XY-8127 Conf Pos Abrir
        [557].S.BITS1.4   // 120-XY-8127 Conf Pos Cerrar
        [557].S.BITS1.29   // 120-XY-8127 Falla Abrir
        [557].S.BITS1.30   // 120-XY-8127 Falla Cerrar
        [557].S.BITS2.20   // 120-XY-8127 Reset Falla
        [557].S.BITS2.23   // 120-XY-8127 Test
        [557].S.BITS2.27   // 120-XY-8127 Cmd. Open
        [557].S.BITS2.30   // 120-XY-8127 OUT CLOSE
        [557].S.BITS2.31   // 120-XY-8127 OUT OPEN
        [558].S.BITS1.0   // 120-TDC-002 Enable
        [558].S.BITS1.1   // 120-TDC-002 Falla Resumen
        [558].S.BITS1.2   // 120-TDC-002 Conf. Marcha
        [558].S.BITS1.4   // 120-TDC-002 Cmd. Automatico
        [558].S.BITS1.26   // 120-TDC-002 FLL
        [558].S.BITS1.27   // 120-TDC-002 FV0
        [558].S.BITS1.28   // 120-TDC-002 FATO
        [558].S.BITS1.30   // 120-TDC-002 Falla Partida
        [558].S.BITS2.27   // 120-TDC-002 Cmd. Marcha
        [558].S.BITS2.20   // 120-TDC-002 Reset Falla
        [558].S.BITS2.23   // 120-TDC-002 Test
        [558].S.BITS2.30   // 120-TDC-002 OUT MARCHA
        [559].S.BITS1.0   // 120-CAN-001 Enable
        [559].S.BITS1.1   // 120-CAN-001 Falla Resumen
        [559].S.BITS1.2   // 120-CAN-001 Conf Pos Abrir
        [559].S.BITS1.4   // 120-CAN-001 Conf Pos Cerrar
        [559].S.BITS1.29   // 120-CAN-001 Falla Abrir
        [559].S.BITS1.30   // 120-CAN-001 Falla Cerrar
        [559].S.BITS2.20   // 120-CAN-001 Reset Falla
        [559].S.BITS2.23   // 120-CAN-001 Test
        [559].S.BITS2.27   // 120-CAN-001 Cmd. Open
        [559].S.BITS2.30   // 120-CAN-001 OUT CLOSE
        [559].S.BITS2.31   // 120-CAN-001 OUT OPEN
        [561].S.BITS1.0   // 110-TDC-003/2 Enable
        [561].S.BITS1.1   // 110-TDC-003/2 Falla Resumen
        [561].S.BITS1.2   // 110-TDC-003/2 Conf. Marcha
        [561].S.BITS1.4   // 110-TDC-003/2 Cmd. Automatico
        [561].S.BITS1.26   // 110-TDC-003/2 FLL
        [561].S.BITS1.27   // 110-TDC-003/2 FV0
        [561].S.BITS1.28   // 110-TDC-003/2 FATO
        [561].S.BITS1.30   // 110-TDC-003/2 Falla Partida
        [561].S.BITS2.27   // 110-TDC-003/2 Cmd. Marcha
        [561].S.BITS2.20   // 110-TDC-003/2 Reset Falla
        [561].S.BITS2.23   // 110-TDC-003/2 Test
        [561].S.BITS2.30   // 110-TDC-003/2 OUT MARCHA
        [562].S.BITS1.0   // 110-TDC-004/2 Enable
        [562].S.BITS1.1   // 110-TDC-004/2 Falla Resumen
        [562].S.BITS1.2   // 110-TDC-004/2 Conf. Marcha
        [562].S.BITS1.4   // 110-TDC-004/2 Cmd. Automatico
        [562].S.BITS1.26   // 110-TDC-004/2 FLL
        [562].S.BITS1.27   // 110-TDC-004/2 FV0
        [562].S.BITS1.28   // 110-TDC-004/2 FATO
        [562].S.BITS1.30   // 110-TDC-004/2 Falla Partida
        [562].S.BITS2.27   // 110-TDC-004/2 Cmd. Marcha
        [562].S.BITS2.20   // 110-TDC-004/2 Reset Falla
        [562].S.BITS2.23   // 110-TDC-004/2 Test
        [562].S.BITS2.30   // 110-TDC-004/2 OUT MARCHA
        [564].S.BITS1.0   // 110-ELV-001/2 Enable
        [564].S.BITS1.1   // 110-ELV-001/2 Falla Resumen
        [564].S.BITS1.2   // 110-ELV-001/2 Conf. Marcha
        [564].S.BITS1.4   // 110-ELV-001/2 Cmd. Automatico
        [564].S.BITS1.26   // 110-ELV-001/2 FLL
        [564].S.BITS1.27   // 110-ELV-001/2 FV0
        [564].S.BITS1.28   // 110-ELV-001/2 FATO
        [564].S.BITS1.30   // 110-ELV-001/2 Falla Partida
        [564].S.BITS2.27   // 110-ELV-001/2 Cmd. Marcha
        [564].S.BITS2.20   // 110-ELV-001/2 Reset Falla
        [564].S.BITS2.23   // 110-ELV-001/2 Test
        [564].S.BITS2.30   // 110-ELV-001/2 OUT MARCHA
        [565].S.BITS1.0   // 120-TDC-001/2 Enable
        [565].S.BITS1.1   // 120-TDC-001/2 Falla Resumen
        [565].S.BITS1.2   // 120-TDC-001/2 Conf. Marcha
        [565].S.BITS1.4   // 120-TDC-001/2 Cmd. Automatico
        [565].S.BITS1.26   // 120-TDC-001/2 FLL
        [565].S.BITS1.27   // 120-TDC-001/2 FV0
        [565].S.BITS1.28   // 120-TDC-001/2 FATO
        [565].S.BITS1.30   // 120-TDC-001/2 Falla Partida
        [565].S.BITS2.27   // 120-TDC-001/2 Cmd. Marcha
        [565].S.BITS2.20   // 120-TDC-001/2 Reset Falla
        [565].S.BITS2.23   // 120-TDC-001/2 Test
        [565].S.BITS2.30   // 120-TDC-001/2 OUT MARCHA
        [566].S.BITS1.0   // 120-HAR-002 Enable
        [566].S.BITS1.1   // 120-HAR-002 Falla Resumen
        [566].S.BITS1.2   // 120-HAR-002 Conf. Marcha
        [566].S.BITS1.4   // 120-HAR-002 Cmd. Automatico
        [566].S.BITS1.26   // 120-HAR-002 FLL
        [566].S.BITS1.27   // 120-HAR-002 FV0
        [566].S.BITS1.28   // 120-HAR-002 FATO
        [566].S.BITS1.30   // 120-HAR-002 Falla Partida
        [566].S.BITS2.27   // 120-HAR-002 Cmd. Marcha
        [566].S.BITS2.20   // 120-HAR-002 Reset Falla
        [566].S.BITS2.23   // 120-HAR-002 Test
        [566].S.BITS2.30   // 120-HAR-002 OUT MARCHA
        [567].S.BITS1.0   // 120-XY-8128 Enable
        [567].S.BITS1.1   // 120-XY-8128 Falla Resumen
        [567].S.BITS1.2   // 120-XY-8128 Conf Pos Abrir
        [567].S.BITS1.4   // 120-XY-8128 Conf Pos Cerrar
        [567].S.BITS1.29   // 120-XY-8128 Falla Abrir
        [567].S.BITS1.30   // 120-XY-8128 Falla Cerrar
        [567].S.BITS2.20   // 120-XY-8128 Reset Falla
        [567].S.BITS2.23   // 120-XY-8128 Test
        [567].S.BITS2.27   // 120-XY-8128 Cmd. Open
        [567].S.BITS2.30   // 120-XY-8128 OUT CLOSE
        [567].S.BITS2.31   // 120-XY-8128 OUT OPEN
        [568].S.BITS1.0   // 120-TDC-003 Enable
        [568].S.BITS1.1   // 120-TDC-003 Falla Resumen
        [568].S.BITS1.2   // 120-TDC-003 Conf. Marcha
        [568].S.BITS1.4   // 120-TDC-003 Cmd. Automatico
        [568].S.BITS1.26   // 120-TDC-003 FLL
        [568].S.BITS1.27   // 120-TDC-003 FV0
        [568].S.BITS1.28   // 120-TDC-003 FATO
        [568].S.BITS1.30   // 120-TDC-003 Falla Partida
        [568].S.BITS2.27   // 120-TDC-003 Cmd. Marcha
        [568].S.BITS2.20   // 120-TDC-003 Reset Falla
        [568].S.BITS2.23   // 120-TDC-003 Test
        [568].S.BITS2.30   // 120-TDC-003 OUT MARCHA
        [569].S.BITS1.0   // 120-CAN-003 Enable
        [569].S.BITS1.1   // 120-CAN-003 Falla Resumen
        [569].S.BITS1.2   // 120-CAN-003 Conf Pos Abrir
        [569].S.BITS1.4   // 120-CAN-003 Conf Pos Cerrar
        [569].S.BITS1.29   // 120-CAN-003 Falla Abrir
        [569].S.BITS1.30   // 120-CAN-003 Falla Cerrar
        [569].S.BITS2.20   // 120-CAN-003 Reset Falla
        [569].S.BITS2.23   // 120-CAN-003 Test
        [569].S.BITS2.27   // 120-CAN-003 Cmd. Open
        [569].S.BITS2.30   // 120-CAN-003 OUT CLOSE
        [569].S.BITS2.31   // 120-CAN-003 OUT OPEN
        [571].S.BITS1.0   // 110-TDC-003/3 Enable
        [571].S.BITS1.1   // 110-TDC-003/3 Falla Resumen
        [571].S.BITS1.2   // 110-TDC-003/3 Conf. Marcha
        [571].S.BITS1.4   // 110-TDC-003/3 Cmd. Automatico
        [571].S.BITS1.26   // 110-TDC-003/3 FLL
        [571].S.BITS1.27   // 110-TDC-003/3 FV0
        [571].S.BITS1.28   // 110-TDC-003/3 FATO
        [571].S.BITS1.30   // 110-TDC-003/3 Falla Partida
        [571].S.BITS2.27   // 110-TDC-003/3 Cmd. Marcha
        [571].S.BITS2.20   // 110-TDC-003/3 Reset Falla
        [571].S.BITS2.23   // 110-TDC-003/3 Test
        [571].S.BITS2.30   // 110-TDC-003/3 OUT MARCHA
        [572].S.BITS1.0   // 110-TDC-004/3 Enable
        [572].S.BITS1.1   // 110-TDC-004/3 Falla Resumen
        [572].S.BITS1.2   // 110-TDC-004/3 Conf. Marcha
        [572].S.BITS1.4   // 110-TDC-004/3 Cmd. Automatico
        [572].S.BITS1.26   // 110-TDC-004/3 FLL
        [572].S.BITS1.27   // 110-TDC-004/3 FV0
        [572].S.BITS1.28   // 110-TDC-004/3 FATO
        [572].S.BITS1.30   // 110-TDC-004/3 Falla Partida
        [572].S.BITS2.27   // 110-TDC-004/3 Cmd. Marcha
        [572].S.BITS2.20   // 110-TDC-004/3 Reset Falla
        [572].S.BITS2.23   // 110-TDC-004/3 Test
        [572].S.BITS2.30   // 110-TDC-004/3 OUT MARCHA
        [573].S.BITS1.0   // 110-TDC-005/3 Enable
        [573].S.BITS1.1   // 110-TDC-005/3 Falla Resumen
        [573].S.BITS1.2   // 110-TDC-005/3 Conf. Marcha
        [573].S.BITS1.4   // 110-TDC-005/3 Cmd. Automatico
        [573].S.BITS1.26   // 110-TDC-005/3 FLL
        [573].S.BITS1.27   // 110-TDC-005/3 FV0
        [573].S.BITS1.28   // 110-TDC-005/3 FATO
        [573].S.BITS1.30   // 110-TDC-005/3 Falla Partida
        [573].S.BITS2.27   // 110-TDC-005/3 Cmd. Marcha
        [573].S.BITS2.20   // 110-TDC-005/3 Reset Falla
        [573].S.BITS2.23   // 110-TDC-005/3 Test
        [573].S.BITS2.30   // 110-TDC-005/3 OUT MARCHA
        [574].S.BITS1.0   // 110-ELV-001/3 Enable
        [574].S.BITS1.1   // 110-ELV-001/3 Falla Resumen
        [574].S.BITS1.2   // 110-ELV-001/3 Conf. Marcha
        [574].S.BITS1.4   // 110-ELV-001/3 Cmd. Automatico
        [574].S.BITS1.26   // 110-ELV-001/3 FLL
        [574].S.BITS1.27   // 110-ELV-001/3 FV0
        [574].S.BITS1.28   // 110-ELV-001/3 FATO
        [574].S.BITS1.30   // 110-ELV-001/3 Falla Partida
        [574].S.BITS2.27   // 110-ELV-001/3 Cmd. Marcha
        [574].S.BITS2.20   // 110-ELV-001/3 Reset Falla
        [574].S.BITS2.23   // 110-ELV-001/3 Test
        [574].S.BITS2.30   // 110-ELV-001/3 OUT MARCHA
        [575].S.BITS1.0   // 120-TDC-001/3 Enable
        [575].S.BITS1.1   // 120-TDC-001/3 Falla Resumen
        [575].S.BITS1.2   // 120-TDC-001/3 Conf. Marcha
        [575].S.BITS1.4   // 120-TDC-001/3 Cmd. Automatico
        [575].S.BITS1.26   // 120-TDC-001/3 FLL
        [575].S.BITS1.27   // 120-TDC-001/3 FV0
        [575].S.BITS1.28   // 120-TDC-001/3 FATO
        [575].S.BITS1.30   // 120-TDC-001/3 Falla Partida
        [575].S.BITS2.27   // 120-TDC-001/3 Cmd. Marcha
        [575].S.BITS2.20   // 120-TDC-001/3 Reset Falla
        [575].S.BITS2.23   // 120-TDC-001/3 Test
        [575].S.BITS2.30   // 120-TDC-001/3 OUT MARCHA
        [576].S.BITS1.0   // 120-HAR-003 Enable
        [576].S.BITS1.1   // 120-HAR-003 Falla Resumen
        [576].S.BITS1.2   // 120-HAR-003 Conf. Marcha
        [576].S.BITS1.4   // 120-HAR-003 Cmd. Automatico
        [576].S.BITS1.26   // 120-HAR-003 FLL
        [576].S.BITS1.27   // 120-HAR-003 FV0
        [576].S.BITS1.28   // 120-HAR-003 FATO
        [576].S.BITS1.30   // 120-HAR-003 Falla Partida
        [576].S.BITS2.27   // 120-HAR-003 Cmd. Marcha
        [576].S.BITS2.20   // 120-HAR-003 Reset Falla
        [576].S.BITS2.23   // 120-HAR-003 Test
        [576].S.BITS2.30   // 120-HAR-003 OUT MARCHA
        [577].S.BITS1.0   // 120-XY-8129 Enable
        [577].S.BITS1.1   // 120-XY-8129 Falla Resumen
        [577].S.BITS1.2   // 120-XY-8129 Conf Pos Abrir
        [577].S.BITS1.4   // 120-XY-8129 Conf Pos Cerrar
        [577].S.BITS1.29   // 120-XY-8129 Falla Abrir
        [577].S.BITS1.30   // 120-XY-8129 Falla Cerrar
        [577].S.BITS2.20   // 120-XY-8129 Reset Falla
        [577].S.BITS2.23   // 120-XY-8129 Test
        [577].S.BITS2.27   // 120-XY-8129 Cmd. Open
        [577].S.BITS2.30   // 120-XY-8129 OUT CLOSE
        [577].S.BITS2.31   // 120-XY-8129 OUT OPEN
        [578].S.BITS1.0   // 120-BIF-001 Enable
        [578].S.BITS1.1   // 120-BIF-001 Falla Resumen
        [578].S.BITS1.2   // 120-BIF-001 Conf. Pos. Izquierda
        [578].S.BITS1.4   // 120-BIF-001 Conf. Pos. Derecha
        [578].S.BITS1.29   // 120-BIF-001 Falla Pos. Izquierda
        [578].S.BITS1.30   // 120-BIF-001 Falla Pos. Derecha
        [578].S.BITS2.20   // 120-BIF-001 Reset Falla
        [578].S.BITS2.23   // 120-BIF-001 Test
        [578].S.BITS2.26   // 120-BIF-001 Cmd. Pos . Izquierda
        [578].S.BITS2.27   // 120-BIF-001 Cmd. Pos. Derecha
        [578].S.BITS2.30   // 120-BIF-001 Out Izquierda
        [578].S.BITS2.31   // 120-BIF-001 Out Derecha
        [581].S.BITS1.0   // 120-TDC-005 Enable
        [581].S.BITS1.1   // 120-TDC-005 Falla Resumen
        [581].S.BITS1.2   // 120-TDC-005 Conf. Marcha
        [581].S.BITS1.4   // 120-TDC-005 Cmd. Automatico
        [581].S.BITS1.26   // 120-TDC-005 FLL
        [581].S.BITS1.27   // 120-TDC-005 FV0
        [581].S.BITS1.28   // 120-TDC-005 FATO
        [581].S.BITS1.30   // 120-TDC-005 Falla Partida
        [581].S.BITS2.27   // 120-TDC-005 Cmd. Marcha
        [581].S.BITS2.20   // 120-TDC-005 Reset Falla
        [581].S.BITS2.23   // 120-TDC-005 Test
        [581].S.BITS2.30   // 120-TDC-005 OUT MARCHA
        [582].S.BITS1.0   // 120-CAN-007 Enable
        [582].S.BITS1.1   // 120-CAN-007 Falla Resumen
        [582].S.BITS1.2   // 120-CAN-007 Conf Pos Abrir
        [582].S.BITS1.4   // 120-CAN-007 Conf Pos Cerrar
        [582].S.BITS1.29   // 120-CAN-007 Falla Abrir
        [582].S.BITS1.30   // 120-CAN-007 Falla Cerrar
        [582].S.BITS2.20   // 120-CAN-007 Reset Falla
        [582].S.BITS2.23   // 120-CAN-007 Test
        [582].S.BITS2.27   // 120-CAN-007 Cmd. Open
        [582].S.BITS2.30   // 120-CAN-007 OUT CLOSE
        [582].S.BITS2.31   // 120-CAN-007 OUT OPEN
        [583].S.BITS1.0   // 120-CAN-008 Enable
        [583].S.BITS1.1   // 120-CAN-008 Falla Resumen
        [583].S.BITS1.2   // 120-CAN-008 Conf Pos Abrir
        [583].S.BITS1.4   // 120-CAN-008 Conf Pos Cerrar
        [583].S.BITS1.29   // 120-CAN-008 Falla Abrir
        [583].S.BITS1.30   // 120-CAN-008 Falla Cerrar
        [583].S.BITS2.20   // 120-CAN-008 Reset Falla
        [583].S.BITS2.23   // 120-CAN-008 Test
        [583].S.BITS2.27   // 120-CAN-008 Cmd. Open
        [583].S.BITS2.30   // 120-CAN-008 OUT CLOSE
        [583].S.BITS2.31   // 120-CAN-008 OUT OPEN
        [584].S.BITS1.0   // 120-CAN-009 Enable
        [584].S.BITS1.1   // 120-CAN-009 Falla Resumen
        [584].S.BITS1.2   // 120-CAN-009 Conf Pos Abrir
        [584].S.BITS1.4   // 120-CAN-009 Conf Pos Cerrar
        [584].S.BITS1.29   // 120-CAN-009 Falla Abrir
        [584].S.BITS1.30   // 120-CAN-009 Falla Cerrar
        [584].S.BITS2.20   // 120-CAN-009 Reset Falla
        [584].S.BITS2.23   // 120-CAN-009 Test
        [584].S.BITS2.27   // 120-CAN-009 Cmd. Open
        [584].S.BITS2.30   // 120-CAN-009 OUT CLOSE
        [584].S.BITS2.31   // 120-CAN-009 OUT OPEN
        [585].S.BITS1.0   // 120-CAN-010 Enable
        [585].S.BITS1.1   // 120-CAN-010 Falla Resumen
        [585].S.BITS1.2   // 120-CAN-010 Conf Pos Abrir
        [585].S.BITS1.4   // 120-CAN-010 Conf Pos Cerrar
        [585].S.BITS1.29   // 120-CAN-010 Falla Abrir
        [585].S.BITS1.30   // 120-CAN-010 Falla Cerrar
        [585].S.BITS2.20   // 120-CAN-010 Reset Falla
        [585].S.BITS2.23   // 120-CAN-010 Test
        [585].S.BITS2.27   // 120-CAN-010 Cmd. Open
        [585].S.BITS2.30   // 120-CAN-010 OUT CLOSE
        [585].S.BITS2.31   // 120-CAN-010 OUT OPEN
        [586].S.BITS1.0   // 120-CAN-011 Enable
        [586].S.BITS1.1   // 120-CAN-011 Falla Resumen
        [586].S.BITS1.2   // 120-CAN-011 Conf Pos Abrir
        [586].S.BITS1.4   // 120-CAN-011 Conf Pos Cerrar
        [586].S.BITS1.29   // 120-CAN-011 Falla Abrir
        [586].S.BITS1.30   // 120-CAN-011 Falla Cerrar
        [586].S.BITS2.20   // 120-CAN-011 Reset Falla
        [586].S.BITS2.23   // 120-CAN-011 Test
        [586].S.BITS2.27   // 120-CAN-011 Cmd. Open
        [586].S.BITS2.30   // 120-CAN-011 OUT CLOSE
        [586].S.BITS2.31   // 120-CAN-011 OUT OPEN
        [587].S.BITS1.0   // 120-CAN-012 Enable
        [587].S.BITS1.1   // 120-CAN-012 Falla Resumen
        [587].S.BITS1.2   // 120-CAN-012 Conf Pos Abrir
        [587].S.BITS1.4   // 120-CAN-012 Conf Pos Cerrar
        [587].S.BITS1.29   // 120-CAN-012 Falla Abrir
        [587].S.BITS1.30   // 120-CAN-012 Falla Cerrar
        [587].S.BITS2.20   // 120-CAN-012 Reset Falla
        [587].S.BITS2.23   // 120-CAN-012 Test
        [587].S.BITS2.27   // 120-CAN-012 Cmd. Open
        [587].S.BITS2.30   // 120-CAN-012 OUT CLOSE
        [587].S.BITS2.31   // 120-CAN-012 OUT OPEN
        [588].S.BITS1.0   // 120-CAN-013 Enable
        [588].S.BITS1.1   // 120-CAN-013 Falla Resumen
        [588].S.BITS1.2   // 120-CAN-013 Conf Pos Abrir
        [588].S.BITS1.4   // 120-CAN-013 Conf Pos Cerrar
        [588].S.BITS1.29   // 120-CAN-013 Falla Abrir
        [588].S.BITS1.30   // 120-CAN-013 Falla Cerrar
        [588].S.BITS2.20   // 120-CAN-013 Reset Falla
        [588].S.BITS2.23   // 120-CAN-013 Test
        [588].S.BITS2.27   // 120-CAN-013 Cmd. Open
        [588].S.BITS2.30   // 120-CAN-013 OUT CLOSE
        [588].S.BITS2.31   // 120-CAN-013 OUT OPEN
        [589].S.BITS1.0   // 120-CAN-014 Enable
        [589].S.BITS1.1   // 120-CAN-014 Falla Resumen
        [589].S.BITS1.2   // 120-CAN-014 Conf Pos Abrir
        [589].S.BITS1.4   // 120-CAN-014 Conf Pos Cerrar
        [589].S.BITS1.29   // 120-CAN-014 Falla Abrir
        [589].S.BITS1.30   // 120-CAN-014 Falla Cerrar
        [589].S.BITS2.20   // 120-CAN-014 Reset Falla
        [589].S.BITS2.23   // 120-CAN-014 Test
        [589].S.BITS2.27   // 120-CAN-014 Cmd. Open
        [589].S.BITS2.30   // 120-CAN-014 OUT CLOSE
        [589].S.BITS2.31   // 120-CAN-014 OUT OPEN
        [590].S.BITS1.0   // 120-CAN-015 Enable
        [590].S.BITS1.1   // 120-CAN-015 Falla Resumen
        [590].S.BITS1.2   // 120-CAN-015 Conf Pos Abrir
        [590].S.BITS1.4   // 120-CAN-015 Conf Pos Cerrar
        [590].S.BITS1.29   // 120-CAN-015 Falla Abrir
        [590].S.BITS1.30   // 120-CAN-015 Falla Cerrar
        [590].S.BITS2.20   // 120-CAN-015 Reset Falla
        [590].S.BITS2.23   // 120-CAN-015 Test
        [590].S.BITS2.27   // 120-CAN-015 Cmd. Open
        [590].S.BITS2.30   // 120-CAN-015 OUT CLOSE
        [590].S.BITS2.31   // 120-CAN-015 OUT OPEN
        [591].S.BITS1.0   // 120-TDC-006 Enable
        [591].S.BITS1.1   // 120-TDC-006 Falla Resumen
        [591].S.BITS1.2   // 120-TDC-006 Conf. Marcha
        [591].S.BITS1.4   // 120-TDC-006 Cmd. Automatico
        [591].S.BITS1.26   // 120-TDC-006 FLL
        [591].S.BITS1.27   // 120-TDC-006 FV0
        [591].S.BITS1.28   // 120-TDC-006 FATO
        [591].S.BITS1.30   // 120-TDC-006 Falla Partida
        [591].S.BITS2.27   // 120-TDC-006 Cmd. Marcha
        [591].S.BITS2.20   // 120-TDC-006 Reset Falla
        [591].S.BITS2.23   // 120-TDC-006 Test
        [591].S.BITS2.30   // 120-TDC-006 OUT MARCHA
        [592].S.BITS1.0   // 120-CAN-027 Enable
        [592].S.BITS1.1   // 120-CAN-027 Falla Resumen
        [592].S.BITS1.2   // 120-CAN-027 Conf Pos Abrir
        [592].S.BITS1.4   // 120-CAN-027 Conf Pos Cerrar
        [592].S.BITS1.29   // 120-CAN-027 Falla Abrir
        [592].S.BITS1.30   // 120-CAN-027 Falla Cerrar
        [592].S.BITS2.20   // 120-CAN-027 Reset Falla
        [592].S.BITS2.23   // 120-CAN-027 Test
        [592].S.BITS2.27   // 120-CAN-027 Cmd. Open
        [592].S.BITS2.30   // 120-CAN-027 OUT CLOSE
        [592].S.BITS2.31   // 120-CAN-027 OUT OPEN
        [593].S.BITS1.0   // 120-CAN-028 Enable
        [593].S.BITS1.1   // 120-CAN-028 Falla Resumen
        [593].S.BITS1.2   // 120-CAN-028 Conf Pos Abrir
        [593].S.BITS1.4   // 120-CAN-028 Conf Pos Cerrar
        [593].S.BITS1.29   // 120-CAN-028 Falla Abrir
        [593].S.BITS1.30   // 120-CAN-028 Falla Cerrar
        [593].S.BITS2.20   // 120-CAN-028 Reset Falla
        [593].S.BITS2.23   // 120-CAN-028 Test
        [593].S.BITS2.27   // 120-CAN-028 Cmd. Open
        [593].S.BITS2.30   // 120-CAN-028 OUT CLOSE
        [593].S.BITS2.31   // 120-CAN-028 OUT OPEN
        [594].S.BITS1.0   // 120-CAN-029 Enable
        [594].S.BITS1.1   // 120-CAN-029 Falla Resumen
        [594].S.BITS1.2   // 120-CAN-029 Conf Pos Abrir
        [594].S.BITS1.4   // 120-CAN-029 Conf Pos Cerrar
        [594].S.BITS1.29   // 120-CAN-029 Falla Abrir
        [594].S.BITS1.30   // 120-CAN-029 Falla Cerrar
        [594].S.BITS2.20   // 120-CAN-029 Reset Falla
        [594].S.BITS2.23   // 120-CAN-029 Test
        [594].S.BITS2.27   // 120-CAN-029 Cmd. Open
        [594].S.BITS2.30   // 120-CAN-029 OUT CLOSE
        [594].S.BITS2.31   // 120-CAN-029 OUT OPEN
        [595].S.BITS1.0   // 120-CAN-030 Enable
        [595].S.BITS1.1   // 120-CAN-030 Falla Resumen
        [595].S.BITS1.2   // 120-CAN-030 Conf Pos Abrir
        [595].S.BITS1.4   // 120-CAN-030 Conf Pos Cerrar
        [595].S.BITS1.29   // 120-CAN-030 Falla Abrir
        [595].S.BITS1.30   // 120-CAN-030 Falla Cerrar
        [595].S.BITS2.20   // 120-CAN-030 Reset Falla
        [595].S.BITS2.23   // 120-CAN-030 Test
        [595].S.BITS2.27   // 120-CAN-030 Cmd. Open
        [595].S.BITS2.30   // 120-CAN-030 OUT CLOSE
        [595].S.BITS2.31   // 120-CAN-030 OUT OPEN
        [596].S.BITS1.0   // 120-CAN-031 Enable
        [596].S.BITS1.1   // 120-CAN-031 Falla Resumen
        [596].S.BITS1.2   // 120-CAN-031 Conf Pos Abrir
        [596].S.BITS1.4   // 120-CAN-031 Conf Pos Cerrar
        [596].S.BITS1.29   // 120-CAN-031 Falla Abrir
        [596].S.BITS1.30   // 120-CAN-031 Falla Cerrar
        [596].S.BITS2.20   // 120-CAN-031 Reset Falla
        [596].S.BITS2.23   // 120-CAN-031 Test
        [596].S.BITS2.27   // 120-CAN-031 Cmd. Open
        [596].S.BITS2.30   // 120-CAN-031 OUT CLOSE
        [596].S.BITS2.31   // 120-CAN-031 OUT OPEN
        [601].S.BITS1.0   // 120-TDC-007 Enable
        [601].S.BITS1.1   // 120-TDC-007 Falla Resumen
        [601].S.BITS1.2   // 120-TDC-007 Conf. Marcha
        [601].S.BITS1.4   // 120-TDC-007 Cmd. Automatico
        [601].S.BITS1.26   // 120-TDC-007 FLL
        [601].S.BITS1.27   // 120-TDC-007 FV0
        [601].S.BITS1.28   // 120-TDC-007 FATO
        [601].S.BITS1.30   // 120-TDC-007 Falla Partida
        [601].S.BITS2.27   // 120-TDC-007 Cmd. Marcha
        [601].S.BITS2.20   // 120-TDC-007 Reset Falla
        [601].S.BITS2.23   // 120-TDC-007 Test
        [601].S.BITS2.30   // 120-TDC-007 OUT MARCHA
        [602].S.BITS1.0   // 120-CAN-039 Enable
        [602].S.BITS1.1   // 120-CAN-039 Falla Resumen
        [602].S.BITS1.2   // 120-CAN-039 Conf Pos Abrir
        [602].S.BITS1.4   // 120-CAN-039 Conf Pos Cerrar
        [602].S.BITS1.29   // 120-CAN-039 Falla Abrir
        [602].S.BITS1.30   // 120-CAN-039 Falla Cerrar
        [602].S.BITS2.20   // 120-CAN-039 Reset Falla
        [602].S.BITS2.23   // 120-CAN-039 Test
        [602].S.BITS2.27   // 120-CAN-039 Cmd. Open
        [602].S.BITS2.30   // 120-CAN-039 OUT CLOSE
        [602].S.BITS2.31   // 120-CAN-039 OUT OPEN
        [603].S.BITS1.0   // 120-CAN-040 Enable
        [603].S.BITS1.1   // 120-CAN-040 Falla Resumen
        [603].S.BITS1.2   // 120-CAN-040 Conf Pos Abrir
        [603].S.BITS1.4   // 120-CAN-040 Conf Pos Cerrar
        [603].S.BITS1.29   // 120-CAN-040 Falla Abrir
        [603].S.BITS1.30   // 120-CAN-040 Falla Cerrar
        [603].S.BITS2.20   // 120-CAN-040 Reset Falla
        [603].S.BITS2.23   // 120-CAN-040 Test
        [603].S.BITS2.27   // 120-CAN-040 Cmd. Open
        [603].S.BITS2.30   // 120-CAN-040 OUT CLOSE
        [603].S.BITS2.31   // 120-CAN-040 OUT OPEN
        [604].S.BITS1.0   // 120-CAN-041 Enable
        [604].S.BITS1.1   // 120-CAN-041 Falla Resumen
        [604].S.BITS1.2   // 120-CAN-041 Conf Pos Abrir
        [604].S.BITS1.4   // 120-CAN-041 Conf Pos Cerrar
        [604].S.BITS1.29   // 120-CAN-041 Falla Abrir
        [604].S.BITS1.30   // 120-CAN-041 Falla Cerrar
        [604].S.BITS2.20   // 120-CAN-041 Reset Falla
        [604].S.BITS2.23   // 120-CAN-041 Test
        [604].S.BITS2.27   // 120-CAN-041 Cmd. Open
        [604].S.BITS2.30   // 120-CAN-041 OUT CLOSE
        [604].S.BITS2.31   // 120-CAN-041 OUT OPEN
        [605].S.BITS1.0   // 120-CAN-042 Enable
        [605].S.BITS1.1   // 120-CAN-042 Falla Resumen
        [605].S.BITS1.2   // 120-CAN-042 Conf Pos Abrir
        [605].S.BITS1.4   // 120-CAN-042 Conf Pos Cerrar
        [605].S.BITS1.29   // 120-CAN-042 Falla Abrir
        [605].S.BITS1.30   // 120-CAN-042 Falla Cerrar
        [605].S.BITS2.20   // 120-CAN-042 Reset Falla
        [605].S.BITS2.23   // 120-CAN-042 Test
        [605].S.BITS2.27   // 120-CAN-042 Cmd. Open
        [605].S.BITS2.30   // 120-CAN-042 OUT CLOSE
        [605].S.BITS2.31   // 120-CAN-042 OUT OPEN
        [606].S.BITS1.0   // 120-CAN-043 Enable
        [606].S.BITS1.1   // 120-CAN-043 Falla Resumen
        [606].S.BITS1.2   // 120-CAN-043 Conf Pos Abrir
        [606].S.BITS1.4   // 120-CAN-043 Conf Pos Cerrar
        [606].S.BITS1.29   // 120-CAN-043 Falla Abrir
        [606].S.BITS1.30   // 120-CAN-043 Falla Cerrar
        [606].S.BITS2.20   // 120-CAN-043 Reset Falla
        [606].S.BITS2.23   // 120-CAN-043 Test
        [606].S.BITS2.27   // 120-CAN-043 Cmd. Open
        [606].S.BITS2.30   // 120-CAN-043 OUT CLOSE
        [606].S.BITS2.31   // 120-CAN-043 OUT OPEN
        [607].S.BITS1.0   // 120-CAN-044 Enable
        [607].S.BITS1.1   // 120-CAN-044 Falla Resumen
        [607].S.BITS1.2   // 120-CAN-044 Conf Pos Abrir
        [607].S.BITS1.4   // 120-CAN-044 Conf Pos Cerrar
        [607].S.BITS1.29   // 120-CAN-044 Falla Abrir
        [607].S.BITS1.30   // 120-CAN-044 Falla Cerrar
        [607].S.BITS2.20   // 120-CAN-044 Reset Falla
        [607].S.BITS2.23   // 120-CAN-044 Test
        [607].S.BITS2.27   // 120-CAN-044 Cmd. Open
        [607].S.BITS2.30   // 120-CAN-044 OUT CLOSE
        [607].S.BITS2.31   // 120-CAN-044 OUT OPEN
        [608].S.BITS1.0   // 120-CAN-045 Enable
        [608].S.BITS1.1   // 120-CAN-045 Falla Resumen
        [608].S.BITS1.2   // 120-CAN-045 Conf Pos Abrir
        [608].S.BITS1.4   // 120-CAN-045 Conf Pos Cerrar
        [608].S.BITS1.29   // 120-CAN-045 Falla Abrir
        [608].S.BITS1.30   // 120-CAN-045 Falla Cerrar
        [608].S.BITS2.20   // 120-CAN-045 Reset Falla
        [608].S.BITS2.23   // 120-CAN-045 Test
        [608].S.BITS2.27   // 120-CAN-045 Cmd. Open
        [608].S.BITS2.30   // 120-CAN-045 OUT CLOSE
        [608].S.BITS2.31   // 120-CAN-045 OUT OPEN
        [611].S.BITS1.0   // 120-TDC-008 Enable
        [611].S.BITS1.1   // 120-TDC-008 Falla Resumen
        [611].S.BITS1.2   // 120-TDC-008 Conf. Marcha
        [611].S.BITS1.4   // 120-TDC-008 Cmd. Automatico
        [611].S.BITS1.26   // 120-TDC-008 FLL
        [611].S.BITS1.27   // 120-TDC-008 FV0
        [611].S.BITS1.28   // 120-TDC-008 FATO
        [611].S.BITS1.30   // 120-TDC-008 Falla Partida
        [611].S.BITS2.27   // 120-TDC-008 Cmd. Marcha
        [611].S.BITS2.20   // 120-TDC-008 Reset Falla
        [611].S.BITS2.23   // 120-TDC-008 Test
        [611].S.BITS2.30   // 120-TDC-008 OUT MARCHA
        [612].S.BITS1.0   // 120-CAN-055 Enable
        [612].S.BITS1.1   // 120-CAN-055 Falla Resumen
        [612].S.BITS1.2   // 120-CAN-055 Conf Pos Abrir
        [612].S.BITS1.4   // 120-CAN-055 Conf Pos Cerrar
        [612].S.BITS1.29   // 120-CAN-055 Falla Abrir
        [612].S.BITS1.30   // 120-CAN-055 Falla Cerrar
        [612].S.BITS2.20   // 120-CAN-055 Reset Falla
        [612].S.BITS2.23   // 120-CAN-055 Test
        [612].S.BITS2.27   // 120-CAN-055 Cmd. Open
        [612].S.BITS2.30   // 120-CAN-055 OUT CLOSE
        [612].S.BITS2.31   // 120-CAN-055 OUT OPEN
        [613].S.BITS1.0   // 120-CAN-056 Enable
        [613].S.BITS1.1   // 120-CAN-056 Falla Resumen
        [613].S.BITS1.2   // 120-CAN-056 Conf Pos Abrir
        [613].S.BITS1.4   // 120-CAN-056 Conf Pos Cerrar
        [613].S.BITS1.29   // 120-CAN-056 Falla Abrir
        [613].S.BITS1.30   // 120-CAN-056 Falla Cerrar
        [613].S.BITS2.20   // 120-CAN-056 Reset Falla
        [613].S.BITS2.23   // 120-CAN-056 Test
        [613].S.BITS2.27   // 120-CAN-056 Cmd. Open
        [613].S.BITS2.30   // 120-CAN-056 OUT CLOSE
        [613].S.BITS2.31   // 120-CAN-056 OUT OPEN
        [614].S.BITS1.0   // 120-CAN-057 Enable
        [614].S.BITS1.1   // 120-CAN-057 Falla Resumen
        [614].S.BITS1.2   // 120-CAN-057 Conf Pos Abrir
        [614].S.BITS1.4   // 120-CAN-057 Conf Pos Cerrar
        [614].S.BITS1.29   // 120-CAN-057 Falla Abrir
        [614].S.BITS1.30   // 120-CAN-057 Falla Cerrar
        [614].S.BITS2.20   // 120-CAN-057 Reset Falla
        [614].S.BITS2.23   // 120-CAN-057 Test
        [614].S.BITS2.27   // 120-CAN-057 Cmd. Open
        [614].S.BITS2.30   // 120-CAN-057 OUT CLOSE
        [614].S.BITS2.31   // 120-CAN-057 OUT OPEN
        [615].S.BITS1.0   // 120-CAN-058 Enable
        [615].S.BITS1.1   // 120-CAN-058 Falla Resumen
        [615].S.BITS1.2   // 120-CAN-058 Conf Pos Abrir
        [615].S.BITS1.4   // 120-CAN-058 Conf Pos Cerrar
        [615].S.BITS1.29   // 120-CAN-058 Falla Abrir
        [615].S.BITS1.30   // 120-CAN-058 Falla Cerrar
        [615].S.BITS2.20   // 120-CAN-058 Reset Falla
        [615].S.BITS2.23   // 120-CAN-058 Test
        [615].S.BITS2.27   // 120-CAN-058 Cmd. Open
        [615].S.BITS2.30   // 120-CAN-058 OUT CLOSE
        [615].S.BITS2.31   // 120-CAN-058 OUT OPEN
        [616].S.BITS1.0   // 120-CAN-059 Enable
        [616].S.BITS1.1   // 120-CAN-059 Falla Resumen
        [616].S.BITS1.2   // 120-CAN-059 Conf Pos Abrir
        [616].S.BITS1.4   // 120-CAN-059 Conf Pos Cerrar
        [616].S.BITS1.29   // 120-CAN-059 Falla Abrir
        [616].S.BITS1.30   // 120-CAN-059 Falla Cerrar
        [616].S.BITS2.20   // 120-CAN-059 Reset Falla
        [616].S.BITS2.23   // 120-CAN-059 Test
        [616].S.BITS2.27   // 120-CAN-059 Cmd. Open
        [616].S.BITS2.30   // 120-CAN-059 OUT CLOSE
        [616].S.BITS2.31   // 120-CAN-059 OUT OPEN
        [617].S.BITS1.0   // 120-CAN-060 Enable
        [617].S.BITS1.1   // 120-CAN-060 Falla Resumen
        [617].S.BITS1.2   // 120-CAN-060 Conf Pos Abrir
        [617].S.BITS1.4   // 120-CAN-060 Conf Pos Cerrar
        [617].S.BITS1.29   // 120-CAN-060 Falla Abrir
        [617].S.BITS1.30   // 120-CAN-060 Falla Cerrar
        [617].S.BITS2.20   // 120-CAN-060 Reset Falla
        [617].S.BITS2.23   // 120-CAN-060 Test
        [617].S.BITS2.27   // 120-CAN-060 Cmd. Open
        [617].S.BITS2.30   // 120-CAN-060 OUT CLOSE
        [617].S.BITS2.31   // 120-CAN-060 OUT OPEN
        [618].S.BITS1.0   // 120-CAN-061 Enable
        [618].S.BITS1.1   // 120-CAN-061 Falla Resumen
        [618].S.BITS1.2   // 120-CAN-061 Conf Pos Abrir
        [618].S.BITS1.4   // 120-CAN-061 Conf Pos Cerrar
        [618].S.BITS1.29   // 120-CAN-061 Falla Abrir
        [618].S.BITS1.30   // 120-CAN-061 Falla Cerrar
        [618].S.BITS2.20   // 120-CAN-061 Reset Falla
        [618].S.BITS2.23   // 120-CAN-061 Test
        [618].S.BITS2.27   // 120-CAN-061 Cmd. Open
        [618].S.BITS2.30   // 120-CAN-061 OUT CLOSE
        [618].S.BITS2.31   // 120-CAN-061 OUT OPEN
        [621].S.BITS1.8   // 120-BIN-001 LL
        [621].S.BITS1.9   // 120-BIN-001 LM
        [621].S.BITS1.10   // 120-BIN-001 LH
        [622].S.BITS1.0   // 120-CAN-017 Enable
        [622].S.BITS1.1   // 120-CAN-017 Falla Resumen
        [622].S.BITS1.2   // 120-CAN-017 Conf Pos Abrir
        [622].S.BITS1.4   // 120-CAN-017 Conf Pos Cerrar
        [622].S.BITS1.29   // 120-CAN-017 Falla Abrir
        [622].S.BITS1.30   // 120-CAN-017 Falla Cerrar
        [622].S.BITS2.20   // 120-CAN-017 Reset Falla
        [622].S.BITS2.23   // 120-CAN-017 Test
        [622].S.BITS2.27   // 120-CAN-017 Cmd. Open
        [622].S.BITS2.30   // 120-CAN-017 OUT CLOSE
        [622].S.BITS2.31   // 120-CAN-017 OUT OPEN
        [623].S.BITS1.8   // 120-BIN-002 LL
        [623].S.BITS1.9   // 120-BIN-002 LM
        [623].S.BITS1.10   // 120-BIN-002 LH
        [624].S.BITS1.0   // 120-CAN-018 Enable
        [624].S.BITS1.1   // 120-CAN-018 Falla Resumen
        [624].S.BITS1.2   // 120-CAN-018 Conf Pos Abrir
        [624].S.BITS1.4   // 120-CAN-018 Conf Pos Cerrar
        [624].S.BITS1.29   // 120-CAN-018 Falla Abrir
        [624].S.BITS1.30   // 120-CAN-018 Falla Cerrar
        [624].S.BITS2.20   // 120-CAN-018 Reset Falla
        [624].S.BITS2.23   // 120-CAN-018 Test
        [624].S.BITS2.27   // 120-CAN-018 Cmd. Open
        [624].S.BITS2.30   // 120-CAN-018 OUT CLOSE
        [624].S.BITS2.31   // 120-CAN-018 OUT OPEN
        [625].S.BITS1.8   // 120-BIN-003 LL
        [625].S.BITS1.9   // 120-BIN-003 LM
        [625].S.BITS1.10   // 120-BIN-003 LH
        [626].S.BITS1.0   // 120-CAN-019 Enable
        [626].S.BITS1.1   // 120-CAN-019 Falla Resumen
        [626].S.BITS1.2   // 120-CAN-019 Conf Pos Abrir
        [626].S.BITS1.4   // 120-CAN-019 Conf Pos Cerrar
        [626].S.BITS1.29   // 120-CAN-019 Falla Abrir
        [626].S.BITS1.30   // 120-CAN-019 Falla Cerrar
        [626].S.BITS2.20   // 120-CAN-019 Reset Falla
        [626].S.BITS2.23   // 120-CAN-019 Test
        [626].S.BITS2.27   // 120-CAN-019 Cmd. Open
        [626].S.BITS2.30   // 120-CAN-019 OUT CLOSE
        [626].S.BITS2.31   // 120-CAN-019 OUT OPEN
        [627].S.BITS1.8   // 120-BIN-004 LL
        [627].S.BITS1.9   // 120-BIN-004 LM
        [627].S.BITS1.10   // 120-BIN-004 LH
        [628].S.BITS1.0   // 120-CAN-020 Enable
        [628].S.BITS1.1   // 120-CAN-020 Falla Resumen
        [628].S.BITS1.2   // 120-CAN-020 Conf Pos Abrir
        [628].S.BITS1.4   // 120-CAN-020 Conf Pos Cerrar
        [628].S.BITS1.29   // 120-CAN-020 Falla Abrir
        [628].S.BITS1.30   // 120-CAN-020 Falla Cerrar
        [628].S.BITS2.20   // 120-CAN-020 Reset Falla
        [628].S.BITS2.23   // 120-CAN-020 Test
        [628].S.BITS2.27   // 120-CAN-020 Cmd. Open
        [628].S.BITS2.30   // 120-CAN-020 OUT CLOSE
        [628].S.BITS2.31   // 120-CAN-020 OUT OPEN
        [629].S.BITS1.8   // 120-BIN-005 LL
        [629].S.BITS1.9   // 120-BIN-005 LM
        [629].S.BITS1.10   // 120-BIN-005 LH
        [630].S.BITS1.0   // 120-CAN-021 Enable
        [630].S.BITS1.1   // 120-CAN-021 Falla Resumen
        [630].S.BITS1.2   // 120-CAN-021 Conf Pos Abrir
        [630].S.BITS1.4   // 120-CAN-021 Conf Pos Cerrar
        [630].S.BITS1.29   // 120-CAN-021 Falla Abrir
        [630].S.BITS1.30   // 120-CAN-021 Falla Cerrar
        [630].S.BITS2.20   // 120-CAN-021 Reset Falla
        [630].S.BITS2.23   // 120-CAN-021 Test
        [630].S.BITS2.27   // 120-CAN-021 Cmd. Open
        [630].S.BITS2.30   // 120-CAN-021 OUT CLOSE
        [630].S.BITS2.31   // 120-CAN-021 OUT OPEN
        [631].S.BITS1.8   // 120-BIN-006 LL
        [631].S.BITS1.9   // 120-BIN-006 LM
        [631].S.BITS1.10   // 120-BIN-006 LH
        [632].S.BITS1.0   // 120-CAN-022 Enable
        [632].S.BITS1.1   // 120-CAN-022 Falla Resumen
        [632].S.BITS1.2   // 120-CAN-022 Conf Pos Abrir
        [632].S.BITS1.4   // 120-CAN-022 Conf Pos Cerrar
        [632].S.BITS1.29   // 120-CAN-022 Falla Abrir
        [632].S.BITS1.30   // 120-CAN-022 Falla Cerrar
        [632].S.BITS2.20   // 120-CAN-022 Reset Falla
        [632].S.BITS2.23   // 120-CAN-022 Test
        [632].S.BITS2.27   // 120-CAN-022 Cmd. Open
        [632].S.BITS2.30   // 120-CAN-022 OUT CLOSE
        [632].S.BITS2.31   // 120-CAN-022 OUT OPEN
        [633].S.BITS1.8   // 120-BIN-007 LL
        [633].S.BITS1.9   // 120-BIN-007 LM
        [633].S.BITS1.10   // 120-BIN-007 LH
        [634].S.BITS1.0   // 120-CAN-023 Enable
        [634].S.BITS1.1   // 120-CAN-023 Falla Resumen
        [634].S.BITS1.2   // 120-CAN-023 Conf Pos Abrir
        [634].S.BITS1.4   // 120-CAN-023 Conf Pos Cerrar
        [634].S.BITS1.29   // 120-CAN-023 Falla Abrir
        [634].S.BITS1.30   // 120-CAN-023 Falla Cerrar
        [634].S.BITS2.20   // 120-CAN-023 Reset Falla
        [634].S.BITS2.23   // 120-CAN-023 Test
        [634].S.BITS2.27   // 120-CAN-023 Cmd. Open
        [634].S.BITS2.30   // 120-CAN-023 OUT CLOSE
        [634].S.BITS2.31   // 120-CAN-023 OUT OPEN
        [635].S.BITS1.8   // 120-BIN-008 LL
        [635].S.BITS1.9   // 120-BIN-008 LM
        [635].S.BITS1.10   // 120-BIN-008 LH
        [636].S.BITS1.0   // 120-CAN-024 Enable
        [636].S.BITS1.1   // 120-CAN-024 Falla Resumen
        [636].S.BITS1.2   // 120-CAN-024 Conf Pos Abrir
        [636].S.BITS1.4   // 120-CAN-024 Conf Pos Cerrar
        [636].S.BITS1.29   // 120-CAN-024 Falla Abrir
        [636].S.BITS1.30   // 120-CAN-024 Falla Cerrar
        [636].S.BITS2.20   // 120-CAN-024 Reset Falla
        [636].S.BITS2.23   // 120-CAN-024 Test
        [636].S.BITS2.27   // 120-CAN-024 Cmd. Open
        [636].S.BITS2.30   // 120-CAN-024 OUT CLOSE
        [636].S.BITS2.31   // 120-CAN-024 OUT OPEN
        [637].S.BITS1.8   // 120-BIN-009 LL
        [637].S.BITS1.9   // 120-BIN-009 LM
        [637].S.BITS1.10   // 120-BIN-009 LH
        [638].S.BITS1.0   // 120-CAN-025 Enable
        [638].S.BITS1.1   // 120-CAN-025 Falla Resumen
        [638].S.BITS1.2   // 120-CAN-025 Conf Pos Abrir
        [638].S.BITS1.4   // 120-CAN-025 Conf Pos Cerrar
        [638].S.BITS1.29   // 120-CAN-025 Falla Abrir
        [638].S.BITS1.30   // 120-CAN-025 Falla Cerrar
        [638].S.BITS2.20   // 120-CAN-025 Reset Falla
        [638].S.BITS2.23   // 120-CAN-025 Test
        [638].S.BITS2.27   // 120-CAN-025 Cmd. Open
        [638].S.BITS2.30   // 120-CAN-025 OUT CLOSE
        [638].S.BITS2.31   // 120-CAN-025 OUT OPEN
        [639].S.BITS1.8   // 120-BIN-010 LL
        [639].S.BITS1.9   // 120-BIN-010 LM
        [639].S.BITS1.10   // 120-BIN-010 LH
        [640].S.BITS1.0   // 120-CAN-026 Enable
        [640].S.BITS1.1   // 120-CAN-026 Falla Resumen
        [640].S.BITS1.2   // 120-CAN-026 Conf Pos Abrir
        [640].S.BITS1.4   // 120-CAN-026 Conf Pos Cerrar
        [640].S.BITS1.29   // 120-CAN-026 Falla Abrir
        [640].S.BITS1.30   // 120-CAN-026 Falla Cerrar
        [640].S.BITS2.20   // 120-CAN-026 Reset Falla
        [640].S.BITS2.23   // 120-CAN-026 Test
        [640].S.BITS2.27   // 120-CAN-026 Cmd. Open
        [640].S.BITS2.30   // 120-CAN-026 OUT CLOSE
        [640].S.BITS2.31   // 120-CAN-026 OUT OPEN
        [641].S.BITS1.8   // 120-BIN-011 LL
        [641].S.BITS1.9   // 120-BIN-011 LM
        [641].S.BITS1.10   // 120-BIN-011 LH
        [642].S.BITS1.0   // 120-CAN-033 Enable
        [642].S.BITS1.1   // 120-CAN-033 Falla Resumen
        [642].S.BITS1.2   // 120-CAN-033 Conf Pos Abrir
        [642].S.BITS1.4   // 120-CAN-033 Conf Pos Cerrar
        [642].S.BITS1.29   // 120-CAN-033 Falla Abrir
        [642].S.BITS1.30   // 120-CAN-033 Falla Cerrar
        [642].S.BITS2.20   // 120-CAN-033 Reset Falla
        [642].S.BITS2.23   // 120-CAN-033 Test
        [642].S.BITS2.27   // 120-CAN-033 Cmd. Open
        [642].S.BITS2.30   // 120-CAN-033 OUT CLOSE
        [642].S.BITS2.31   // 120-CAN-033 OUT OPEN
        [643].S.BITS1.8   // 120-BIN-012 LL
        [643].S.BITS1.9   // 120-BIN-012 LM
        [643].S.BITS1.10   // 120-BIN-012 LH
        [644].S.BITS1.0   // 120-CAN-034 Enable
        [644].S.BITS1.1   // 120-CAN-034 Falla Resumen
        [644].S.BITS1.2   // 120-CAN-034 Conf Pos Abrir
        [644].S.BITS1.4   // 120-CAN-034 Conf Pos Cerrar
        [644].S.BITS1.29   // 120-CAN-034 Falla Abrir
        [644].S.BITS1.30   // 120-CAN-034 Falla Cerrar
        [644].S.BITS2.20   // 120-CAN-034 Reset Falla
        [644].S.BITS2.23   // 120-CAN-034 Test
        [644].S.BITS2.27   // 120-CAN-034 Cmd. Open
        [644].S.BITS2.30   // 120-CAN-034 OUT CLOSE
        [644].S.BITS2.31   // 120-CAN-034 OUT OPEN
        [645].S.BITS1.8   // 120-BIN-013 LL
        [645].S.BITS1.9   // 120-BIN-013 LM
        [645].S.BITS1.10   // 120-BIN-013 LH
        [646].S.BITS1.0   // 120-CAN-035 Enable
        [646].S.BITS1.1   // 120-CAN-035 Falla Resumen
        [646].S.BITS1.2   // 120-CAN-035 Conf Pos Abrir
        [646].S.BITS1.4   // 120-CAN-035 Conf Pos Cerrar
        [646].S.BITS1.29   // 120-CAN-035 Falla Abrir
        [646].S.BITS1.30   // 120-CAN-035 Falla Cerrar
        [646].S.BITS2.20   // 120-CAN-035 Reset Falla
        [646].S.BITS2.23   // 120-CAN-035 Test
        [646].S.BITS2.27   // 120-CAN-035 Cmd. Open
        [646].S.BITS2.30   // 120-CAN-035 OUT CLOSE
        [646].S.BITS2.31   // 120-CAN-035 OUT OPEN
        [647].S.BITS1.8   // 120-BIN-014 LL
        [647].S.BITS1.9   // 120-BIN-014 LM
        [647].S.BITS1.10   // 120-BIN-014 LH
        [648].S.BITS1.0   // 120-CAN-036 Enable
        [648].S.BITS1.1   // 120-CAN-036 Falla Resumen
        [648].S.BITS1.2   // 120-CAN-036 Conf Pos Abrir
        [648].S.BITS1.4   // 120-CAN-036 Conf Pos Cerrar
        [648].S.BITS1.29   // 120-CAN-036 Falla Abrir
        [648].S.BITS1.30   // 120-CAN-036 Falla Cerrar
        [648].S.BITS2.20   // 120-CAN-036 Reset Falla
        [648].S.BITS2.23   // 120-CAN-036 Test
        [648].S.BITS2.27   // 120-CAN-036 Cmd. Open
        [648].S.BITS2.30   // 120-CAN-036 OUT CLOSE
        [648].S.BITS2.31   // 120-CAN-036 OUT OPEN
        [649].S.BITS1.8   // 120-BIN-015 LL
        [649].S.BITS1.9   // 120-BIN-015 LM
        [649].S.BITS1.10   // 120-BIN-015 LH
        [650].S.BITS1.0   // 120-CAN-037 Enable
        [650].S.BITS1.1   // 120-CAN-037 Falla Resumen
        [650].S.BITS1.2   // 120-CAN-037 Conf Pos Abrir
        [650].S.BITS1.4   // 120-CAN-037 Conf Pos Cerrar
        [650].S.BITS1.29   // 120-CAN-037 Falla Abrir
        [650].S.BITS1.30   // 120-CAN-037 Falla Cerrar
        [650].S.BITS2.20   // 120-CAN-037 Reset Falla
        [650].S.BITS2.23   // 120-CAN-037 Test
        [650].S.BITS2.27   // 120-CAN-037 Cmd. Open
        [650].S.BITS2.30   // 120-CAN-037 OUT CLOSE
        [650].S.BITS2.31   // 120-CAN-037 OUT OPEN
        [651].S.BITS1.8   // 120-BIN-016 LL
        [651].S.BITS1.9   // 120-BIN-016 LM
        [651].S.BITS1.10   // 120-BIN-016 LH
        [652].S.BITS1.0   // 120-CAN-038 Enable
        [652].S.BITS1.1   // 120-CAN-038 Falla Resumen
        [652].S.BITS1.2   // 120-CAN-038 Conf Pos Abrir
        [652].S.BITS1.4   // 120-CAN-038 Conf Pos Cerrar
        [652].S.BITS1.29   // 120-CAN-038 Falla Abrir
        [652].S.BITS1.30   // 120-CAN-038 Falla Cerrar
        [652].S.BITS2.20   // 120-CAN-038 Reset Falla
        [652].S.BITS2.23   // 120-CAN-038 Test
        [652].S.BITS2.27   // 120-CAN-038 Cmd. Open
        [652].S.BITS2.30   // 120-CAN-038 OUT CLOSE
        [652].S.BITS2.31   // 120-CAN-038 OUT OPEN
        [653].S.BITS1.8   // 120-BIN-017 LL
        [653].S.BITS1.9   // 120-BIN-017 LM
        [653].S.BITS1.10   // 120-BIN-017 LH
        [654].S.BITS1.0   // 120-CAN-047 Enable
        [654].S.BITS1.1   // 120-CAN-047 Falla Resumen
        [654].S.BITS1.2   // 120-CAN-047 Conf Pos Abrir
        [654].S.BITS1.4   // 120-CAN-047 Conf Pos Cerrar
        [654].S.BITS1.29   // 120-CAN-047 Falla Abrir
        [654].S.BITS1.30   // 120-CAN-047 Falla Cerrar
        [654].S.BITS2.20   // 120-CAN-047 Reset Falla
        [654].S.BITS2.23   // 120-CAN-047 Test
        [654].S.BITS2.27   // 120-CAN-047 Cmd. Open
        [654].S.BITS2.30   // 120-CAN-047 OUT CLOSE
        [654].S.BITS2.31   // 120-CAN-047 OUT OPEN
        [655].S.BITS1.8   // 120-BIN-018 LL
        [655].S.BITS1.9   // 120-BIN-018 LM
        [655].S.BITS1.10   // 120-BIN-018 LH
        [656].S.BITS1.0   // 120-CAN-048 Enable
        [656].S.BITS1.1   // 120-CAN-048 Falla Resumen
        [656].S.BITS1.2   // 120-CAN-048 Conf Pos Abrir
        [656].S.BITS1.4   // 120-CAN-048 Conf Pos Cerrar
        [656].S.BITS1.29   // 120-CAN-048 Falla Abrir
        [656].S.BITS1.30   // 120-CAN-048 Falla Cerrar
        [656].S.BITS2.20   // 120-CAN-048 Reset Falla
        [656].S.BITS2.23   // 120-CAN-048 Test
        [656].S.BITS2.27   // 120-CAN-048 Cmd. Open
        [656].S.BITS2.30   // 120-CAN-048 OUT CLOSE
        [656].S.BITS2.31   // 120-CAN-048 OUT OPEN
        [657].S.BITS1.8   // 120-BIN-019 LL
        [657].S.BITS1.9   // 120-BIN-019 LM
        [657].S.BITS1.10   // 120-BIN-019 LH
        [658].S.BITS1.0   // 120-CAN-049 Enable
        [658].S.BITS1.1   // 120-CAN-049 Falla Resumen
        [658].S.BITS1.2   // 120-CAN-049 Conf Pos Abrir
        [658].S.BITS1.4   // 120-CAN-049 Conf Pos Cerrar
        [658].S.BITS1.29   // 120-CAN-049 Falla Abrir
        [658].S.BITS1.30   // 120-CAN-049 Falla Cerrar
        [658].S.BITS2.20   // 120-CAN-049 Reset Falla
        [658].S.BITS2.23   // 120-CAN-049 Test
        [658].S.BITS2.27   // 120-CAN-049 Cmd. Open
        [658].S.BITS2.30   // 120-CAN-049 OUT CLOSE
        [658].S.BITS2.31   // 120-CAN-049 OUT OPEN
        [659].S.BITS1.8   // 120-BIN-020 LL
        [659].S.BITS1.9   // 120-BIN-020 LM
        [659].S.BITS1.10   // 120-BIN-020 LH
        [660].S.BITS1.0   // 120-CAN-050 Enable
        [660].S.BITS1.1   // 120-CAN-050 Falla Resumen
        [660].S.BITS1.2   // 120-CAN-050 Conf Pos Abrir
        [660].S.BITS1.4   // 120-CAN-050 Conf Pos Cerrar
        [660].S.BITS1.29   // 120-CAN-050 Falla Abrir
        [660].S.BITS1.30   // 120-CAN-050 Falla Cerrar
        [660].S.BITS2.20   // 120-CAN-050 Reset Falla
        [660].S.BITS2.23   // 120-CAN-050 Test
        [660].S.BITS2.27   // 120-CAN-050 Cmd. Open
        [660].S.BITS2.30   // 120-CAN-050 OUT CLOSE
        [660].S.BITS2.31   // 120-CAN-050 OUT OPEN
        [661].S.BITS1.8   // 120-BIN-021 LL
        [661].S.BITS1.9   // 120-BIN-021 LM
        [661].S.BITS1.10   // 120-BIN-021 LH
        [662].S.BITS1.0   // 120-CAN-051 Enable
        [662].S.BITS1.1   // 120-CAN-051 Falla Resumen
        [662].S.BITS1.2   // 120-CAN-051 Conf Pos Abrir
        [662].S.BITS1.4   // 120-CAN-051 Conf Pos Cerrar
        [662].S.BITS1.29   // 120-CAN-051 Falla Abrir
        [662].S.BITS1.30   // 120-CAN-051 Falla Cerrar
        [662].S.BITS2.20   // 120-CAN-051 Reset Falla
        [662].S.BITS2.23   // 120-CAN-051 Test
        [662].S.BITS2.27   // 120-CAN-051 Cmd. Open
        [662].S.BITS2.30   // 120-CAN-051 OUT CLOSE
        [662].S.BITS2.31   // 120-CAN-051 OUT OPEN
        [663].S.BITS1.8   // 120-BIN-022 LL
        [663].S.BITS1.9   // 120-BIN-022 LM
        [663].S.BITS1.10   // 120-BIN-022 LH
        [664].S.BITS1.0   // 120-CAN-052 Enable
        [664].S.BITS1.1   // 120-CAN-052 Falla Resumen
        [664].S.BITS1.2   // 120-CAN-052 Conf Pos Abrir
        [664].S.BITS1.4   // 120-CAN-052 Conf Pos Cerrar
        [664].S.BITS1.29   // 120-CAN-052 Falla Abrir
        [664].S.BITS1.30   // 120-CAN-052 Falla Cerrar
        [664].S.BITS2.20   // 120-CAN-052 Reset Falla
        [664].S.BITS2.23   // 120-CAN-052 Test
        [664].S.BITS2.27   // 120-CAN-052 Cmd. Open
        [664].S.BITS2.30   // 120-CAN-052 OUT CLOSE
        [664].S.BITS2.31   // 120-CAN-052 OUT OPEN
        [665].S.BITS1.8   // 120-BIN-023 LL
        [665].S.BITS1.9   // 120-BIN-023 LM
        [665].S.BITS1.10   // 120-BIN-023 LH
        [666].S.BITS1.0   // 120-CAN-053 Enable
        [666].S.BITS1.1   // 120-CAN-053 Falla Resumen
        [666].S.BITS1.2   // 120-CAN-053 Conf Pos Abrir
        [666].S.BITS1.4   // 120-CAN-053 Conf Pos Cerrar
        [666].S.BITS1.29   // 120-CAN-053 Falla Abrir
        [666].S.BITS1.30   // 120-CAN-053 Falla Cerrar
        [666].S.BITS2.20   // 120-CAN-053 Reset Falla
        [666].S.BITS2.23   // 120-CAN-053 Test
        [666].S.BITS2.27   // 120-CAN-053 Cmd. Open
        [666].S.BITS2.30   // 120-CAN-053 OUT CLOSE
        [666].S.BITS2.31   // 120-CAN-053 OUT OPEN
        [667].S.BITS1.8   // 120-BIN-024 LL
        [667].S.BITS1.9   // 120-BIN-024 LM
        [667].S.BITS1.10   // 120-BIN-024 LH
        [668].S.BITS1.0   // 120-CAN-054 Enable
        [668].S.BITS1.1   // 120-CAN-054 Falla Resumen
        [668].S.BITS1.2   // 120-CAN-054 Conf Pos Abrir
        [668].S.BITS1.4   // 120-CAN-054 Conf Pos Cerrar
        [668].S.BITS1.29   // 120-CAN-054 Falla Abrir
        [668].S.BITS1.30   // 120-CAN-054 Falla Cerrar
        [668].S.BITS2.20   // 120-CAN-054 Reset Falla
        [668].S.BITS2.23   // 120-CAN-054 Test
        [668].S.BITS2.27   // 120-CAN-054 Cmd. Open
        [668].S.BITS2.30   // 120-CAN-054 OUT CLOSE
        [668].S.BITS2.31   // 120-CAN-054 OUT OPEN
        [669].S.BITS1.8   // 120-BIN-025 LL
        [669].S.BITS1.9   // 120-BIN-025 LM
        [669].S.BITS1.10   // 120-BIN-025 LH
        [670].S.BITS1.0   // 120-CAN-063 Enable
        [670].S.BITS1.1   // 120-CAN-063 Falla Resumen
        [670].S.BITS1.2   // 120-CAN-063 Conf Pos Abrir
        [670].S.BITS1.4   // 120-CAN-063 Conf Pos Cerrar
        [670].S.BITS1.29   // 120-CAN-063 Falla Abrir
        [670].S.BITS1.30   // 120-CAN-063 Falla Cerrar
        [670].S.BITS2.20   // 120-CAN-063 Reset Falla
        [670].S.BITS2.23   // 120-CAN-063 Test
        [670].S.BITS2.27   // 120-CAN-063 Cmd. Open
        [670].S.BITS2.30   // 120-CAN-063 OUT CLOSE
        [670].S.BITS2.31   // 120-CAN-063 OUT OPEN
        [671].S.BITS1.8   // 120-BIN-026 LL
        [671].S.BITS1.9   // 120-BIN-026 LM
        [671].S.BITS1.10   // 120-BIN-026 LH
        [672].S.BITS1.0   // 120-CAN-064 Enable
        [672].S.BITS1.1   // 120-CAN-064 Falla Resumen
        [672].S.BITS1.2   // 120-CAN-064 Conf Pos Abrir
        [672].S.BITS1.4   // 120-CAN-064 Conf Pos Cerrar
        [672].S.BITS1.29   // 120-CAN-064 Falla Abrir
        [672].S.BITS1.30   // 120-CAN-064 Falla Cerrar
        [672].S.BITS2.20   // 120-CAN-064 Reset Falla
        [672].S.BITS2.23   // 120-CAN-064 Test
        [672].S.BITS2.27   // 120-CAN-064 Cmd. Open
        [672].S.BITS2.30   // 120-CAN-064 OUT CLOSE
        [672].S.BITS2.31   // 120-CAN-064 OUT OPEN
        [673].S.BITS1.8   // 120-BIN-027 LL
        [673].S.BITS1.9   // 120-BIN-027 LM
        [673].S.BITS1.10   // 120-BIN-027 LH
        [674].S.BITS1.0   // 120-CAN-065 Enable
        [674].S.BITS1.1   // 120-CAN-065 Falla Resumen
        [674].S.BITS1.2   // 120-CAN-065 Conf Pos Abrir
        [674].S.BITS1.4   // 120-CAN-065 Conf Pos Cerrar
        [674].S.BITS1.29   // 120-CAN-065 Falla Abrir
        [674].S.BITS1.30   // 120-CAN-065 Falla Cerrar
        [674].S.BITS2.20   // 120-CAN-065 Reset Falla
        [674].S.BITS2.23   // 120-CAN-065 Test
        [674].S.BITS2.27   // 120-CAN-065 Cmd. Open
        [674].S.BITS2.30   // 120-CAN-065 OUT CLOSE
        [674].S.BITS2.31   // 120-CAN-065 OUT OPEN
        [675].S.BITS1.8   // 120-BIN-028 LL
        [675].S.BITS1.9   // 120-BIN-028 LM
        [675].S.BITS1.10   // 120-BIN-028 LH
        [676].S.BITS1.0   // 120-CAN-066 Enable
        [676].S.BITS1.1   // 120-CAN-066 Falla Resumen
        [676].S.BITS1.2   // 120-CAN-066 Conf Pos Abrir
        [676].S.BITS1.4   // 120-CAN-066 Conf Pos Cerrar
        [676].S.BITS1.29   // 120-CAN-066 Falla Abrir
        [676].S.BITS1.30   // 120-CAN-066 Falla Cerrar
        [676].S.BITS2.20   // 120-CAN-066 Reset Falla
        [676].S.BITS2.23   // 120-CAN-066 Test
        [676].S.BITS2.27   // 120-CAN-066 Cmd. Open
        [676].S.BITS2.30   // 120-CAN-066 OUT CLOSE
        [676].S.BITS2.31   // 120-CAN-066 OUT OPEN
        [117].S.BITS1.9   // 7-BIN-1116 LM
        [117].S.BITS1.10   // 7-BIN-1116 LH
        [164].S.BITS1.9   // 7-BIN-1163 LM
        [164].S.BITS1.10   // 7-BIN-1163 LH
        [165].S.BITS1.9   // 100-BIF-003 Conf. Pos Izquierda
        [165].S.BITS1.10   // 100-BIF-003 Conf. Pos Derecha
        [199].S.BITS1.10   // 100-TOR-009 Velocidad Cero
        [205].S.BITS1.10   // 100-TOR-036 Velocidad Cero
        [208].S.BITS1.10   // 100-TOR-012 Velocidad Cero
        [214].S.BITS1.10   // 7-ETQ-1179a LH
        [218].S.BITS1.10   // 100-TOR-038 Velocidad Cero
        [239].S.BITS1.10   // 100-MMA-001 Velocidad Cero
        [242].S.BITS1.10   // 100-TOR-021 Velocidad Cero
        [244].S.BITS1.10   // 100-TOR-020 Velocidad Cero
        [248].S.BITS1.10   // 100-TOR-018 Velocidad Cero
        [255].S.BITS1.9   // 100-TOL-004-1 Conf. Cerrado
        [255].S.BITS1.10   // 100-TOL-004-1 Conf. Abierto
        [264].S.BITS1.10   // 100-DOS-001-MO2 Velocidad Cero
        [268].S.BITS1.10   // 100-DOS-001-M04 Velocidad Cero
        [272].S.BITS1.10   // 100-DOS-001-M06 Velocidad Cero
        [274].S.BITS1.10   // 100-DOS-001-M07 Velocidad Cero
        [278].S.BITS1.10   // 100-DOS-001-M09 Velocidad Cero
        [280].S.BITS1.10   // 100-DOS-100-M10 Velocidad Cero
        [289].S.BITS1.10   // 100-TDP-003 Velocidad Cero
        [292].S.BITS1.10   // 100-TDP-004 Velocidad Cero
        [293].S.BITS1.10   // 100-ELV-002 Velocidad Cero
        [294].S.BITS1.10   // 100-TDP-005 Velocidad Cero
        [299].S.BITS1.10   // 100-TDP-006 Velocidad Cero
        [302].S.BITS1.10   // 100-BCE-003 Velocidad Cero
        [304].S.BITS1.10   // 100-BCE-005 Velocidad Cero
        [312].S.BITS1.10   // 100-BCE-001 Velocidad Cero
        [314].S.BITS1.10   // 100-VEN-ACORG-1 Velocidad Cero
        [315].S.BITS1.10   // 100-VEN-ACORG-2 Velocidad Cero
        [316].S.BITS1.9   // 8-ENF-630 LM
        [316].S.BITS1.10   // 8-ENF-630 LH
        [317].S.BITS1.9   // 100-VEN-COLINA-1 Sobrecarga
        [317].S.BITS1.10   // 100-VEN-COLINA-1 Velocidad Cero
        [322].S.BITS1.10   // 100-MIX-001-M Velocidad Cero
        [323].S.BITS1.10   // 100-VIB-001 Velocidad Cero
        [325].S.BITS1.10   // 100-TDC-007 Velocidad Cero
        [326].S.BITS1.10   // 8-ENF-640 LH
        [332].S.BITS1.10   // 110-FIL-001 Velocidad Cero
        [334].S.BITS1.10   // 110-FIL-002 Velocidad Cero
        [336].S.BITS1.10   // 110-FIL-003 Velocidad Cero
        [337].S.BITS1.10   // 110-VEN-003 Velocidad Cero
        [342].S.BITS1.10   // 110-TDC-001 Velocidad Cero
        [344].S.BITS1.9   // 110-LMG-001-01 Conf. Cerrado
        [344].S.BITS1.10   // 110-LMG-001-01 Conf. Abierto
        [346].S.BITS1.9   // 110-LMG-002 Conf. Pos Izquierda
        [346].S.BITS1.10   // 110-LMG-002 Conf. Pos Derecha
        [349].S.BITS1.10   // 8-TOL-712 LH
        [351].S.BITS1.10   // 110-TOR-005 Velocidad Cero
        [363].S.BITS1.9   // 110-CAN-008/1 Conf. Cerrado
        [363].S.BITS1.10   // 110-CAN-008/1 Conf. Abierto
        [364].S.BITS1.9   // 110-CAN-009/1 Conf. Cerrado
        [364].S.BITS1.10   // 110-CAN-009/1 Conf. Abierto
        [365].S.BITS1.10   // 110-CAN-010/1 Velocidad Cero
        [370].S.BITS1.10   // 110-TOR-001/1 Velocidad Cero
        [372].S.BITS1.10   // 110-ACD-001/1 Velocidad Cero
        [373].S.BITS1.10   // 110-EXP-001/1 Velocidad Cero
        [374].S.BITS1.10   // 110-DES-001/1 Velocidad Cero
        [375].S.BITS1.10   // 110-CAE-001/1 Velocidad Cero
        [376].S.BITS1.10   // 110-PLT-001/1 Velocidad Cero
        [377].S.BITS1.9   // 110-BIF-001/1 Conf. Pos Izquierda
        [377].S.BITS1.10   // 110-BIF-001/1 Conf. Pos Derecha
        [381].S.BITS1.10   // 110-ESC-001/1 Velocidad Cero
        [382].S.BITS1.10   // 110-ENF-001/1-4 Velocidad Cero
        [384].S.BITS1.10   // 110-ENF-001/1-1 Velocidad Cero
        [387].S.BITS1.10   // 110-ESC-003/1 Velocidad Cero
        [389].S.BITS1.10   // 110-VAL-001/1-1 Velocidad Cero
        [390].S.BITS1.10   // 110-VEN-001/1-1 Velocidad Cero
        [391].S.BITS1.10   // 110-ENF-001/1-5 Velocidad Cero
        [401].S.BITS1.10   // 110-ESC-002/1 Velocidad Cero
        [402].S.BITS1.10   // 110-ENF-002/1-4 Velocidad Cero
        [404].S.BITS1.10   // 110-ENF-002/1-1 Velocidad Cero
        [407].S.BITS1.10   // 110-ESC-004/1 Velocidad Cero
        [409].S.BITS1.10   // 110-VAL-002/1-1 Velocidad Cero
        [410].S.BITS1.10   // 110-VEN-002/1-1 Velocidad Cero
        [411].S.BITS1.10   // 110-ENF-002/1-5 Velocidad Cero
        [414].S.BITS1.10   // 110-TOR-002/1 Velocidad Cero
        [415].S.BITS1.10   // 110-TOR-003/1 Velocidad Cero
        [416].S.BITS1.10   // 110-ELV-002/1 Velocidad Cero
        [417].S.BITS1.10   // 110-TOL-006/1 Velocidad Cero
        [418].S.BITS1.10   // 110-TOR-004/1 Velocidad Cero
        [423].S.BITS1.9   // 110-CAN-008/2 Conf. Cerrado
        [423].S.BITS1.10   // 110-CAN-008/2 Conf. Abierto
        [424].S.BITS1.9   // 110-CAN-009/2 Conf. Cerrado
        [424].S.BITS1.10   // 110-CAN-009/2 Conf. Abierto
        [425].S.BITS1.10   // 110-CAN-010/2 Velocidad Cero
        [430].S.BITS1.10   // 110-TOR-001/2 Velocidad Cero
        [432].S.BITS1.10   // 110-ACD-001/2 Velocidad Cero
        [433].S.BITS1.10   // 110-EXP-001/2 Velocidad Cero
        [434].S.BITS1.10   // 110-DES-001/2 Velocidad Cero
        [435].S.BITS1.10   // 110-CAE-001/2 Velocidad Cero
        [436].S.BITS1.10   // 110-PLT-001/2 Velocidad Cero
        [437].S.BITS1.9   // 110-BIF-001/2 Conf. Pos Izquierda
        [437].S.BITS1.10   // 110-BIF-001/2 Conf. Pos Derecha
        [441].S.BITS1.10   // 110-ESC-001/2 Velocidad Cero
        [442].S.BITS1.10   // 9-BIN-704 LH
        [444].S.BITS1.10   // 9-BIN-706 LH
        [447].S.BITS1.10   // 110-ESC-003/2 Velocidad Cero
        [449].S.BITS1.10   // 110-VAL-001/2-1 Velocidad Cero
        [450].S.BITS1.10   // 9-BIN-712 LH
        [451].S.BITS1.10   // 110-ENF-001/2-5 Velocidad Cero
        [461].S.BITS1.10   // 110-ESC-002/2 Velocidad Cero
        [462].S.BITS1.10   // 9-BIN-724 LH
        [464].S.BITS1.10   // 9-BIN-726 LH
        [467].S.BITS1.10   // 110-ESC-004/2 Velocidad Cero
        [469].S.BITS1.10   // 110-VAL-002/2-1 Velocidad Cero
        [470].S.BITS1.10   // 110-VEN-002/2 Velocidad Cero
        [471].S.BITS1.10   // 110-ENF-002/2-5 Velocidad Cero
        [474].S.BITS1.10   // 110-TOR-002/2 Velocidad Cero
        [475].S.BITS1.10   // 110-TOR-003/2 Velocidad Cero
        [476].S.BITS1.10   // 110-ELV-002/2 Velocidad Cero
        [478].S.BITS1.10   // 110-TOR-004/2 Velocidad Cero
        [493].S.BITS1.9   // 110-CAN-008/3 Conf. Cerrado
        [493].S.BITS1.10   // 110-CAN-008/3 Conf. Abierto
        [494].S.BITS1.9   // 110-CAN-009/3 Conf. Cerrado
        [495].S.BITS1.10   // 110-CAN-010/3 Velocidad Cero
        [497].S.BITS1.9   // 110-CAN-011/3 Conf. Cerrado
        [497].S.BITS1.10   // 110-CAN-011/3 Conf. Abierto
        [500].S.BITS1.10   // 110-TOR-001/3 Velocidad Cero
        [502].S.BITS1.10   // 110-ACD-001/3 Velocidad Cero
        [503].S.BITS1.10   // 110-EXP-001/3 Velocidad Cero
        [506].S.BITS1.10   // 110-PLT-001/3 Velocidad Cero
        [507].S.BITS1.9   // 110-BIF-001/3 Conf. Pos Izquierda
        [511].S.BITS1.10   // 110-ESC-001/3 Velocidad Cero
        [512].S.BITS1.10   // 110-ENF-001/3-4 Velocidad Cero
        [514].S.BITS1.10   // 110-ENF-001/3-1 Velocidad Cero
        [517].S.BITS1.10   // 110-ESC-003/3 Velocidad Cero
        [519].S.BITS1.10   // 110-VAL-001/3-1 Velocidad Cero
        [520].S.BITS1.10   // 110-VEN-001/3 Velocidad Cero
        [521].S.BITS1.10   // 110-ENF-001/3-5 Velocidad Cero
        [523].S.BITS1.10   // 110-QUE-001-1 Velocidad Cero
        [524].S.BITS1.10   // 110-QUE-001-2 Velocidad Cero
        [531].S.BITS1.10   // 110-ESC-002/3 Velocidad Cero
        [532].S.BITS1.10   // 110-ENF-002/3-4 Velocidad Cero
        [534].S.BITS1.10   // 110-ENF-002/3-1 Velocidad Cero
        [537].S.BITS1.10   // 110-ESC-004/3 Velocidad Cero
        [539].S.BITS1.10   // 110-VEN-002/3-1 Velocidad Cero
        [540].S.BITS1.10   // 110-VEN-002/3 Velocidad Cero
        [541].S.BITS1.10   // 110-ENF-002/3-5 Velocidad Cero
        [544].S.BITS1.10   // 110-TOR-002/3 Velocidad Cero
        [545].S.BITS1.10   // 110-TOR-003/3 Velocidad Cero
        [546].S.BITS1.10   // 110-ELV-002/3 Velocidad Cero
        [548].S.BITS1.10   // 110-TOR-004/3 Velocidad Cero
        [551].S.BITS1.10   // 110-TDC-003/1 Velocidad Cero
        [552].S.BITS1.10   // 110-TDC-004/1 Velocidad Cero
        [554].S.BITS1.10   // 110-ELV-001/1 Velocidad Cero
        [555].S.BITS1.10   // 120-TDC-001/1 Velocidad Cero
        [556].S.BITS1.10   // 120-HAR-001 Velocidad Cero
        [558].S.BITS1.10   // 120-TDC-002 Velocidad Cero
        [561].S.BITS1.10   // 110-TDC-003/2 Velocidad Cero
        [562].S.BITS1.10   // 110-TDC-004/2 Velocidad Cero
        [564].S.BITS1.10   // 110-ELV-001/2 Velocidad Cero
        [565].S.BITS1.10   // 120-TDC-001/2 Velocidad Cero
        [566].S.BITS1.10   // 120-HAR-002 Velocidad Cero
        [568].S.BITS1.10   // 120-TDC-003 Velocidad Cero
        [571].S.BITS1.10   // 110-TDC-003/3 Velocidad Cero
        [572].S.BITS1.10   // 110-TDC-004/3 Velocidad Cero
        [573].S.BITS1.10   // 110-TDC-005/3 Velocidad Cero
        [574].S.BITS1.10   // 110-ELV-001/3 Velocidad Cero
        [575].S.BITS1.10   // 120-TDC-001/3 Velocidad Cero
        [576].S.BITS1.10   // 120-HAR-003 Velocidad Cero
        [578].S.BITS1.9   // 120-BIF-001 Conf. Pos Izquierda
        [578].S.BITS1.10   // 120-BIF-001 Conf. Pos Derecha
        [581].S.BITS1.10   // 120-TDC-005 Velocidad Cero
        [591].S.BITS1.10   // 120-TDC-006 Velocidad Cero
        [601].S.BITS1.10   // 120-TDC-007 Velocidad Cero
        [611].S.BITS1.10   // 120-TDC-008 Velocidad Cero
        [618].S.BITS1.10   // 120-CAN-061 Conf. Abierto
        [622].S.BITS1.10   // 120-CAN-017 Conf. Abierto
        [624].S.BITS1.10   // 120-CAN-018 Conf. Abierto
        [626].S.BITS1.10   // 120-CAN-019 Conf. Abierto
        [628].S.BITS1.10   // 120-CAN-020 Conf. Abierto
        [630].S.BITS1.10   // 120-CAN-021 Conf. Abierto
        [632].S.BITS1.10   // 120-CAN-022 Conf. Abierto
        [634].S.BITS1.10   // 120-CAN-023 Conf. Abierto
        [636].S.BITS1.10   // 120-CAN-024 Conf. Abierto
        [638].S.BITS1.10   // 120-CAN-025 Conf. Abierto
        [640].S.BITS1.10   // 120-CAN-026 Conf. Abierto
        [642].S.BITS1.10   // 120-CAN-033 Conf. Abierto
        [644].S.BITS1.10   // 120-CAN-034 Conf. Abierto
        [646].S.BITS1.10   // 120-CAN-035 Conf. Abierto
        [648].S.BITS1.10   // 120-CAN-036 Conf. Abierto
        [650].S.BITS1.10   // 120-CAN-037 Conf. Abierto
        [652].S.BITS1.10   // 120-CAN-038 Conf. Abierto
        [654].S.BITS1.10   // 120-CAN-047 Conf. Abierto
        [656].S.BITS1.10   // 120-CAN-048 Conf. Abierto
        [658].S.BITS1.10   // 120-CAN-049 Conf. Abierto
        [660].S.BITS1.10   // 120-CAN-050 Conf. Abierto
        [662].S.BITS1.10   // 120-CAN-051 Conf. Abierto
        [664].S.BITS1.10   // 120-CAN-052 Conf. Abierto
        [666].S.BITS1.10   // 120-CAN-053 Conf. Abierto
        [668].S.BITS1.10   // 120-CAN-054 Conf. Abierto
        [670].S.BITS1.10   // 120-CAN-063 Conf. Abierto
        [672].S.BITS1.10   // 120-CAN-064 Conf. Abierto
        [674].S.BITS1.10   // 120-CAN-065 Conf. Abierto
        [676].S.BITS1.10   // 120-CAN-066 Conf. Abierto
        [678].S.BITS1.2   // 120-CAN-067 Conf Pos Abrir
        [678].S.BITS1.4   // 120-CAN-067 Conf Pos Cerrar
        [678].S.BITS1.10   // 120-CAN-067 Conf. Abierto
        [680].S.BITS1.2   // 120-CAN-068 Conf Pos Abrir
        [680].S.BITS1.4   // 120-CAN-068 Conf Pos Cerrar
        [680].S.BITS1.10   // 120-CAN-068 Conf. Abierto
        [682].S.BITS1.2   // 120-CAN-069 Conf Pos Abrir
        [682].S.BITS1.4   // 120-CAN-069 Conf Pos Cerrar
        [682].S.BITS1.10   // 120-CAN-069 Conf. Abierto
        [684].S.BITS1.2   // 120-CAN-070 Conf Pos Abrir
        [684].S.BITS1.4   // 120-CAN-070 Conf Pos Cerrar
        [684].S.BITS1.10   // 120-CAN-070 Conf. Abierto
        [233].S.BITS1.2   // 7-LMG-1187 Conf Pos Abrir
        [233].S.BITS1.4   // 7-LMG-1187 Conf Pos Cerrar
        [234].S.BITS1.2   // 100-CAN-023 Conf Pos Abrir
        [234].S.BITS1.4   // 100-CAN-023 Conf Pos Cerrar
        [235].S.BITS1.2   // 7-LRT-1189 Conf. Marcha
        [235].S.BITS1.4   // 7-LRT-1189 Cmd. Automatico
        [236].S.BITS1.2   // 100-CAN-025 Conf Pos Abrir
        [236].S.BITS1.4   // 100-CAN-025 Conf Pos Cerrar
        [264].S.BITS2.31   // 100-DOS-001-MO2 OUT MARCHA
        [266].S.BITS2.31   // 100-DOS-001-M03 OUT MARCHA
        [270].S.BITS2.31   // 100-DOS-001-M05 OUT MARCHA
        [272].S.BITS2.31   // 100-DOS-001-M06 OUT MARCHA
        [274].S.BITS2.31   // 100-DOS-001-M07 OUT MARCHA
        [276].S.BITS2.31   // 100-DOS-001-M08 OUT MARCHA
        [278].S.BITS2.31   // 100-DOS-001-M09 OUT MARCHA
        [280].S.BITS2.31   // 100-DOS-100-M10 OUT MARCHA
        [282].S.BITS2.31   // 100-DOS-100-M11 OUT MARCHA
        [284].S.BITS2.31   // 100-DOS-100-M12 OUT MARCHA
        [288].S.BITS1.1   // 100-DOS-001-C Falla Resumen
        [288].S.BITS1.2   // 100-DOS-001-C Conf Pos Abrir
        [288].S.BITS1.4   // 100-DOS-001-C Conf Pos Cerrar
        [288].S.BITS1.29   // 100-DOS-001-C Falla Abrir
        [288].S.BITS1.30   // 100-DOS-001-C Falla Cerrar
        [288].S.BITS2.20   // 100-DOS-001-C Reset Falla
        [297].S.BITS1.1   // 100-TOL-003-1 Falla Resumen
        [297].S.BITS1.2   // 100-TOL-003-1 Conf Pos Abrir
        [297].S.BITS1.4   // 100-TOL-003-1 Conf Pos Cerrar
        [297].S.BITS1.29   // 100-TOL-003-1 Falla Abrir
        [297].S.BITS1.30   // 100-TOL-003-1 Falla Cerrar
        [297].S.BITS2.20   // 100-TOL-003-1 Reset Falla
        [314].S.BITS2.31   // 100-VEN-ACORG-1 OUT MARCHA
        [315].S.BITS2.31   // 100-VEN-ACORG-2 OUT MARCHA
        [316].S.BITS2.31   // 100-VEN-LICINA-1 OUT MARCHA
        [384].S.BITS2.31   // 8-CON-764b OUT OPEN
        [385].S.BITS1.1   // 110-ENF-001/1-2 Falla Resumen
        [385].S.BITS1.2   // 110-ENF-001/1-2 Conf Pos Abrir
        [385].S.BITS1.4   // 110-ENF-001/1-2 Conf Pos Cerrar
        [385].S.BITS1.29   // 110-ENF-001/1-2 Falla Abrir
        [385].S.BITS1.30   // 110-ENF-001/1-2 Falla Cerrar
        [385].S.BITS2.20   // 110-ENF-001/1-2 Reset Falla
        [385].S.BITS2.27   // 110-ENF-001/1-2 Cmd. Open
        [385].S.BITS2.30   // 110-ENF-001/1-2 OUT CLOSE
        [387].S.BITS2.31   // 9-CON-651 OUT OPEN
        [391].S.BITS2.31   // 110-ENF-001/1-5 OUT MARCHA
        [402].S.BITS2.31   // 9-CON-664 OUT OPEN
        [404].S.BITS2.31   // 9-CON-666 OUT OPEN
        [405].S.BITS1.1   // 9-CON-667 Falla Resumen
        [405].S.BITS1.2   // 9-CON-667 Conf Pos Abrir
        [405].S.BITS1.4   // 9-CON-667 Conf Pos Cerrar
        [405].S.BITS1.29   // 9-CON-667 Falla Abrir
        [405].S.BITS1.30   // 9-CON-667 Falla Cerrar
        [405].S.BITS2.20   // 9-CON-667 Reset Falla
        [405].S.BITS2.27   // 9-CON-667 Cmd. Open
        [405].S.BITS2.30   // 9-CON-667 OUT CLOSE
        [405].S.BITS2.31   // 9-CON-667 OUT OPEN
        [407].S.BITS2.31   // 110-ESC-004/1 OUT MARCHA
        [411].S.BITS2.31   // 9-CON-673 OUT OPEN
        [414].S.BITS2.31   // 9-CON-676 OUT OPEN
        [418].S.BITS2.31   // 110-TOR-004/1 OUT MARCHA
        [425].S.BITS2.31   // 9-CON-687 OUT OPEN
        [430].S.BITS2.31   // 9-CON-692 OUT OPEN
        [433].S.BITS2.31   // 9-CON-695 OUT OPEN
        [436].S.BITS2.31   // 9-CON-698 OUT OPEN
        [442].S.BITS2.31   // 110-ENF-001/2-4 OUT MARCHA
        [444].S.BITS2.31   // 110-ENF-001/2-1 OUT MARCHA
        [445].S.BITS1.1   // 9-CON-707 Falla Resumen
        [445].S.BITS1.2   // 9-CON-707 Conf Pos Abrir
        [445].S.BITS1.4   // 9-CON-707 Conf Pos Cerrar
        [445].S.BITS1.29   // 9-CON-707 Falla Abrir
        [445].S.BITS1.30   // 9-CON-707 Falla Cerrar
        [445].S.BITS2.20   // 9-CON-707 Reset Falla
